REGION Network 14: PackML Event - Alarms Not Cleared
   RUNG wire#powerrail
      #instStatusAlarmsNotReset(EnableIn := wire#w1, Cfg_Event := "StatusCfg".Event[1], Cfg_MessagePrefix := "MessagePrefix".UN.Alarm, In_EventStatus := "UN".Status, Sts_Active => #instStatusAlarmsNotReset.Sts_Active, Sts_Latched => #instStatusAlarmsNotReset.Sts_Latched)
   END_RUNG
   RUNG wire#powerrail
      Contact( "PackML".Sts.State.Resetting )
      I_Contact( "UN".PackML_Sts_Alarm.sts_Resetting_SC )
   END_RUNG wire#w1
   RUNG wire#powerrail
      Contact( "PackML".Sts.State.Clearing )
      I_Contact( "UN".PackML_Sts_Alarm.sts_Clearing_SC )
   END_RUNG wire#w1
   // the same network as SCL:
   #instStatusAlarmsNotReset(EnableIn := ("PackML".Sts.State.Resetting AND NOT "UN".PackML_Sts_Alarm.sts_Resetting_SC) OR ("PackML".Sts.State.Clearing AND NOT "UN".PackML_Sts_Alarm.sts_Clearing_SC),   // "CPG_Event"
                           Cfg_Event := "StatusCfg".Event[1],
                           Cfg_MessagePrefix := "MessagePrefix".UN.Alarm,
                           In_EventStatus := "UN".Status,
                           Sts_Active => #instStatusAlarmsNotReset.Sts_Active,
                           Sts_Latched => #instStatusAlarmsNotReset.Sts_Latched);
END_REGION

REGION Network 15: Start Command
   // "PackTags".Command.CntrlCmd = 2 (start command value)
   RUNG wire#powerrail
      Contact( "PackML".remoteCommandEnable )
      { S7_Templates := "SrcType := DInt" } EQ_Contact(in1 := "PackTags".Command.CntrlCmd, in2 := "LPMLV30_CMD_START")
      Contact( "PackTags".Command.CmdChangeRequest )
      Coil( "UN".PackML_Sts_Alarm.cmd_Start )
   END_RUNG
   // the same network as SCL:
   "UN".PackML_Sts_Alarm.cmd_Start := "PackML".remoteCommandEnable AND ("PackTags".Command.CntrlCmd = "LPMLV30_CMD_START") AND "PackTags".Command.CmdChangeRequest;
END_REGION

REGION Network 16: Reset Command
   // "PackTags".Command.CntrlCmd = 1 (reset command value)
   RUNG wire#powerrail
      Contact( "PackML".remoteCommandEnable )
      { S7_Templates := "SrcType := DInt" } EQ_Contact(in1 := "PackTags".Command.CntrlCmd, in2 := "LPMLV30_CMD_RESET")
      Contact( "PackTags".Command.CmdChangeRequest )
      Coil( "UN".PackML_Sts_Alarm.cmd_Reset )
   END_RUNG
   // the same network as SCL:
   "UN".PackML_Sts_Alarm.cmd_Reset := "PackML".remoteCommandEnable AND ("PackTags".Command.CntrlCmd = "LPMLV30_CMD_RESET") AND "PackTags".Command.CmdChangeRequest;
END_REGION

REGION Network 17: Clear Command
   // "PackTags".Command.CntrlCmd = 9 (clear command value)
   RUNG wire#powerrail
      Contact( "PackML".remoteCommandEnable )
      { S7_Templates := "SrcType := DInt" } EQ_Contact(in1 := "PackTags".Command.CntrlCmd, in2 := "LPMLV30_CMD_CLEAR")
      Contact( "PackTags".Command.CmdChangeRequest )
      Coil( "UN".PackML_Sts_Alarm.cmd_Clear )
   END_RUNG
   // the same network as SCL:
   "UN".PackML_Sts_Alarm.cmd_Clear := "PackML".remoteCommandEnable AND ("PackTags".Command.CntrlCmd = "LPMLV30_CMD_CLEAR") AND "PackTags".Command.CmdChangeRequest;
END_REGION

REGION Network 18: *** EVENT CONTROL MANAGERS ***
END_REGION

REGION Network 19: Reset Command - for all event managers
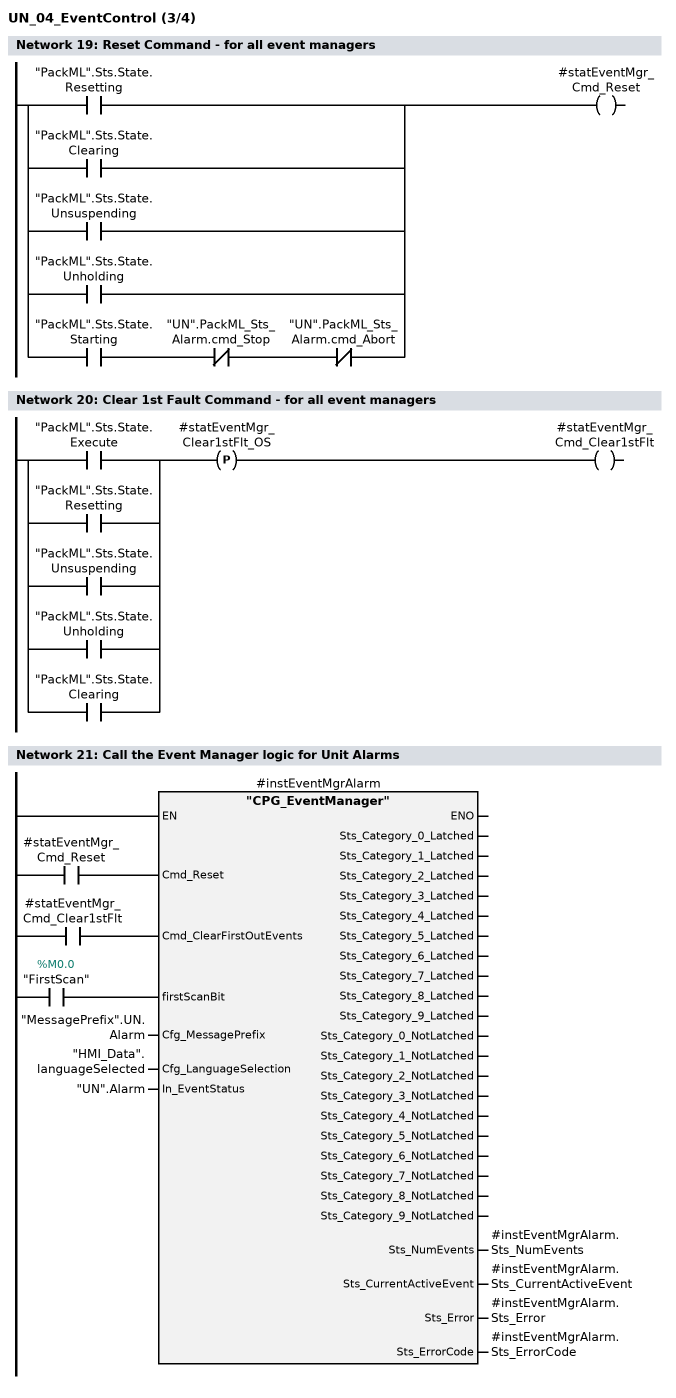
   RUNG wire#powerrail
      Contact( "PackML".Sts.State.Resetting )
      wire#w1
      Coil( #statEventMgr_Cmd_Reset )
   END_RUNG
   RUNG wire#powerrail
      Contact( "PackML".Sts.State.Clearing )
   END_RUNG wire#w1
   RUNG wire#powerrail
      Contact( "PackML".Sts.State.Unsuspending )
   END_RUNG wire#w1
   RUNG wire#powerrail
      Contact( "PackML".Sts.State.Unholding )
   END_RUNG wire#w1
   RUNG wire#powerrail
      Contact( "PackML".Sts.State.Starting )
      I_Contact( "UN".PackML_Sts_Alarm.cmd_Stop )
      I_Contact( "UN".PackML_Sts_Alarm.cmd_Abort )
   END_RUNG wire#w1
   // the same network as SCL:
   #statEventMgr_Cmd_Reset := "PackML".Sts.State.Resetting OR "PackML".Sts.State.Clearing OR "PackML".Sts.State.Unsuspending OR "PackML".Sts.State.Unholding OR ("PackML".Sts.State.Starting AND NOT "UN".PackML_Sts_Alarm.cmd_Stop AND NOT "UN".PackML_Sts_Alarm.cmd_Abort);
END_REGION

REGION Network 20: Clear 1st Fault Command - for all event managers
   RUNG wire#powerrail
      Contact( "PackML".Sts.State.Execute )
      wire#w1
      P_Trig( #statEventMgr_Clear1stFlt_OS )
      Coil( #statEventMgr_Cmd_Clear1stFlt )
   END_RUNG
   RUNG wire#powerrail
      Contact( "PackML".Sts.State.Resetting )
   END_RUNG wire#w1
   RUNG wire#powerrail
      Contact( "PackML".Sts.State.Unsuspending )
   END_RUNG wire#w1
   RUNG wire#powerrail
      Contact( "PackML".Sts.State.Unholding )
   END_RUNG wire#w1
   RUNG wire#powerrail
      Contact( "PackML".Sts.State.Clearing )
   END_RUNG wire#w1
   // the same network as SCL:
   #_w1 := "PackML".Sts.State.Execute OR "PackML".Sts.State.Resetting OR "PackML".Sts.State.Unsuspending OR "PackML".Sts.State.Unholding OR "PackML".Sts.State.Clearing;
   #_w2 := #_w1 AND NOT #statEventMgr_Clear1stFlt_OS;   // rising edge
   #statEventMgr_Clear1stFlt_OS := #_w1;
   #statEventMgr_Cmd_Clear1stFlt := #_w2;
END_REGION

REGION Network 21: Call the Event Manager logic for Unit Alarms
   RUNG wire#powerrail
      #instEventMgrAlarm(Cmd_Reset := wire#w1, Cmd_ClearFirstOutEvents := wire#w2, firstScanBit := wire#w3, Cfg_MessagePrefix := "MessagePrefix".UN.Alarm, Cfg_LanguageSelection := "HMI_Data".languageSelected, In_EventStatus := "UN".Alarm, Sts_Category_0_Latched =>, Sts_Category_1_Latched =>, Sts_Category_2_Latched =>, Sts_Category_3_Latched =>, Sts_Category_4_Latched =>, Sts_Category_5_Latched =>, Sts_Category_6_Latched =>, Sts_Category_7_Latched =>, Sts_Category_8_Latched =>, Sts_Category_9_Latched =>, Sts_Category_0_NotLatched =>, Sts_Category_1_NotLatched =>, Sts_Category_2_NotLatched =>, Sts_Category_3_NotLatched =>, Sts_Category_4_NotLatched =>, Sts_Category_5_NotLatched =>, Sts_Category_6_NotLatched =>, Sts_Category_7_NotLatched =>, Sts_Category_8_NotLatched =>, Sts_Category_9_NotLatched =>, Sts_NumEvents => #instEventMgrAlarm.Sts_NumEvents, Sts_CurrentActiveEvent => #instEventMgrAlarm.Sts_CurrentActiveEvent, Sts_Error => #instEventMgrAlarm.Sts_Error, Sts_ErrorCode => #instEventMgrAlarm.Sts_ErrorCode)
   END_RUNG
   RUNG wire#powerrail
      Contact( #statEventMgr_Cmd_Reset )
   END_RUNG wire#w1
   RUNG wire#powerrail
      Contact( #statEventMgr_Cmd_Clear1stFlt )
   END_RUNG wire#w2
   RUNG wire#powerrail
      Contact( "FirstScan" )
   END_RUNG wire#w3
   // the same network as SCL:
   #instEventMgrAlarm(Cmd_Reset := #statEventMgr_Cmd_Reset,   // "CPG_EventManager"
                      Cmd_ClearFirstOutEvents := #statEventMgr_Cmd_Clear1stFlt,
                      firstScanBit := "FirstScan",
                      Cfg_MessagePrefix := "MessagePrefix".UN.Alarm,
                      Cfg_LanguageSelection := "HMI_Data".languageSelected,
                      In_EventStatus := "UN".Alarm,
                      Sts_NumEvents => #instEventMgrAlarm.Sts_NumEvents,
                      Sts_CurrentActiveEvent => #instEventMgrAlarm.Sts_CurrentActiveEvent,
                      Sts_Error => #instEventMgrAlarm.Sts_Error,
                      Sts_ErrorCode => #instEventMgrAlarm.Sts_ErrorCode);
END_REGION

REGION Network 22: Call the Event Manager logic for Unit Warnings
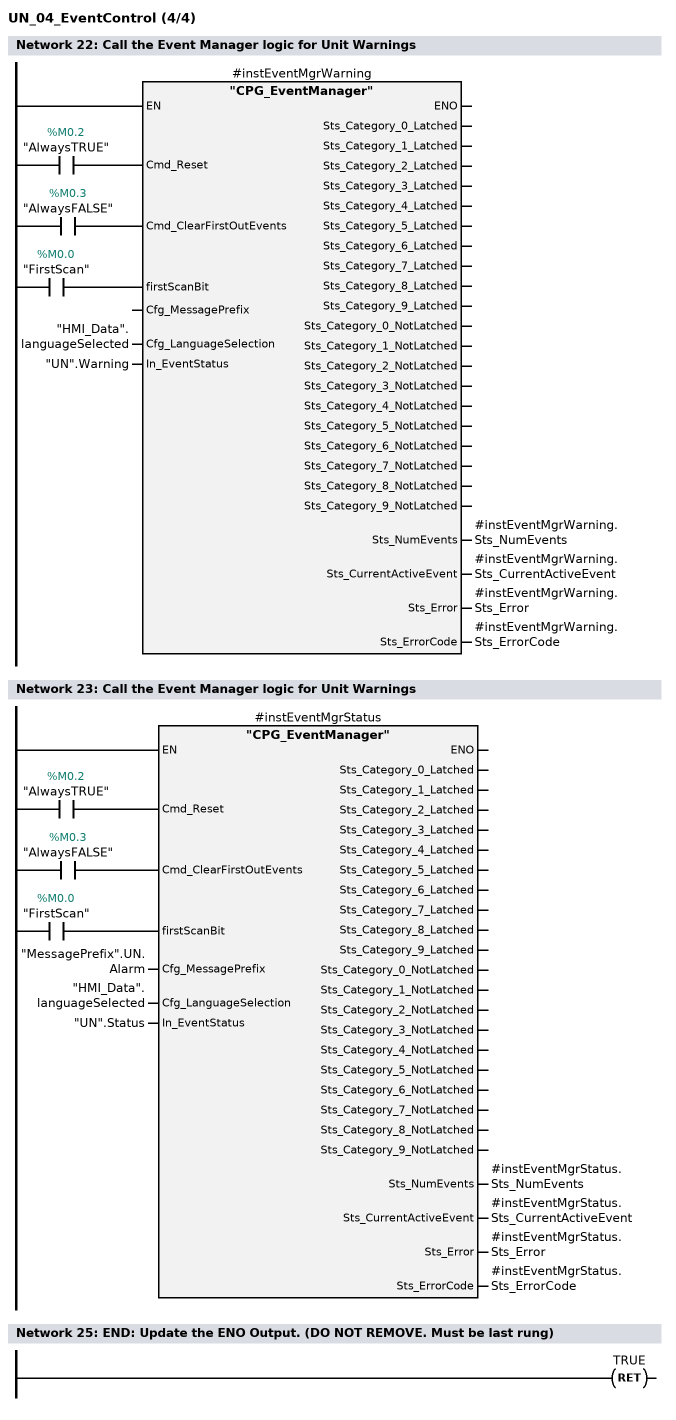
   RUNG wire#powerrail
      #instEventMgrWarning(Cmd_Reset := wire#w1, Cmd_ClearFirstOutEvents := wire#w2, firstScanBit := wire#w3, Cfg_MessagePrefix :=, Cfg_LanguageSelection := "HMI_Data".languageSelected, In_EventStatus := "UN".Warning, Sts_Category_0_Latched =>, Sts_Category_1_Latched =>, Sts_Category_2_Latched =>, Sts_Category_3_Latched =>, Sts_Category_4_Latched =>, Sts_Category_5_Latched =>, Sts_Category_6_Latched =>, Sts_Category_7_Latched =>, Sts_Category_8_Latched =>, Sts_Category_9_Latched =>, Sts_Category_0_NotLatched =>, Sts_Category_1_NotLatched =>, Sts_Category_2_NotLatched =>, Sts_Category_3_NotLatched =>, Sts_Category_4_NotLatched =>, Sts_Category_5_NotLatched =>, Sts_Category_6_NotLatched =>, Sts_Category_7_NotLatched =>, Sts_Category_8_NotLatched =>, Sts_Category_9_NotLatched =>, Sts_NumEvents => #instEventMgrWarning.Sts_NumEvents, Sts_CurrentActiveEvent => #instEventMgrWarning.Sts_CurrentActiveEvent, Sts_Error => #instEventMgrWarning.Sts_Error, Sts_ErrorCode => #instEventMgrWarning.Sts_ErrorCode)
   END_RUNG
   RUNG wire#powerrail
      Contact( "AlwaysTRUE" )
   END_RUNG wire#w1
   RUNG wire#powerrail
      Contact( "AlwaysFALSE" )
   END_RUNG wire#w2
   RUNG wire#powerrail
      Contact( "FirstScan" )
   END_RUNG wire#w3
   // the same network as SCL:
   #instEventMgrWarning(Cmd_Reset := "AlwaysTRUE",   // "CPG_EventManager"
                        Cmd_ClearFirstOutEvents := "AlwaysFALSE",
                        firstScanBit := "FirstScan",
                        Cfg_LanguageSelection := "HMI_Data".languageSelected,
                        In_EventStatus := "UN".Warning,
                        Sts_NumEvents => #instEventMgrWarning.Sts_NumEvents,
                        Sts_CurrentActiveEvent => #instEventMgrWarning.Sts_CurrentActiveEvent,
                        Sts_Error => #instEventMgrWarning.Sts_Error,
                        Sts_ErrorCode => #instEventMgrWarning.Sts_ErrorCode);
END_REGION

REGION Network 23: Call the Event Manager logic for Unit Warnings
   RUNG wire#powerrail
      #instEventMgrStatus(Cmd_Reset := wire#w1, Cmd_ClearFirstOutEvents := wire#w2, firstScanBit := wire#w3, Cfg_MessagePrefix := "MessagePrefix".UN.Alarm, Cfg_LanguageSelection := "HMI_Data".languageSelected, In_EventStatus := "UN".Status, Sts_Category_0_Latched =>, Sts_Category_1_Latched =>, Sts_Category_2_Latched =>, Sts_Category_3_Latched =>, Sts_Category_4_Latched =>, Sts_Category_5_Latched =>, Sts_Category_6_Latched =>, Sts_Category_7_Latched =>, Sts_Category_8_Latched =>, Sts_Category_9_Latched =>, Sts_Category_0_NotLatched =>, Sts_Category_1_NotLatched =>, Sts_Category_2_NotLatched =>, Sts_Category_3_NotLatched =>, Sts_Category_4_NotLatched =>, Sts_Category_5_NotLatched =>, Sts_Category_6_NotLatched =>, Sts_Category_7_NotLatched =>, Sts_Category_8_NotLatched =>, Sts_Category_9_NotLatched =>, Sts_NumEvents => #instEventMgrStatus.Sts_NumEvents, Sts_CurrentActiveEvent => #instEventMgrStatus.Sts_CurrentActiveEvent, Sts_Error => #instEventMgrStatus.Sts_Error, Sts_ErrorCode => #instEventMgrStatus.Sts_ErrorCode)
   END_RUNG
   RUNG wire#powerrail
      Contact( "AlwaysTRUE" )
   END_RUNG wire#w1
   RUNG wire#powerrail
      Contact( "AlwaysFALSE" )
   END_RUNG wire#w2
   RUNG wire#powerrail
      Contact( "FirstScan" )
   END_RUNG wire#w3
   // the same network as SCL:
   #instEventMgrStatus(Cmd_Reset := "AlwaysTRUE",   // "CPG_EventManager"
                       Cmd_ClearFirstOutEvents := "AlwaysFALSE",
                       firstScanBit := "FirstScan",
                       Cfg_MessagePrefix := "MessagePrefix".UN.Alarm,
                       Cfg_LanguageSelection := "HMI_Data".languageSelected,
                       In_EventStatus := "UN".Status,
                       Sts_NumEvents => #instEventMgrStatus.Sts_NumEvents,
                       Sts_CurrentActiveEvent => #instEventMgrStatus.Sts_CurrentActiveEvent,
                       Sts_Error => #instEventMgrStatus.Sts_Error,
                       Sts_ErrorCode => #instEventMgrStatus.Sts_ErrorCode);
END_REGION

REGION Network 25: END: Update the ENO Output. (DO NOT REMOVE. Must be last rung)
   RUNG wire#powerrail
      ReturnCoil( TRUE )
   END_RUNG
   // the same network as SCL:
   ENO := TRUE;
   RETURN;
END_REGION
END_FUNCTION_BLOCK

FUNCTION "CPG_ModuleInitialize" : Void
TITLE = CPG_ModuleInitialize
{ S7_Optimized_Access := 'TRUE' }
AUTHOR : 'tech.team.motioncontrol@siemens.com'
FAMILY : CPG
VERSION : 1.0
//Support: tech.team.motioncontrol@siemens.com
   VAR_INPUT 
      enableIn : Bool;   // Enable the FB call.
      firstScanBit : Bool;   // Bit used to tell logic that this is the first scan of PLC
   END_VAR

   VAR_IN_OUT 
      PackML_ModuleStatus : "CPG_typePackML_ModuleSts";   // PackML Module Status UDT
   END_VAR


BEGIN
	//============================================================================================================
	// SIEMENS AG
	// (c)Copyright 2018 All Rights Reserved
	//------------------------------------------------------------------------------------------------------------
	// Project: CPG Template
	// Tested with: S7-1500 with FW version V2.1
	// Engineering: TIA Portal V14
	// Restrictions: ---
	// Requirements: S7-1500
	// Functionality: This FC will initialize the "PackML" "Status" AND commands within a control module to ensure that the bits are in the correct state IF they are NOT being
	//                used later by that same control module. FOR example, if a start command is NOT being used by a control module, that bit should be turned off TO prevent
	//                unintentional starting OF the machine (in CASE it was accidentally OR through a rung edit turned on). IF a state complete bit FOR a particular state is
	//                NOT being used, that bit should be turned on TO allow the machine TO leave that state. This instruction is NOT needed FOR equipment modules OR the unit
	//                machine since all PackML status AND command bits are programmed in the summation routines.
	// Support: tech.team.motioncontrol@siemens.com
	//------------------------------------------------------------------------------------------------------------
	// Change log table:
	// Version       Date               Expert in charge    Changes applied
	//  01.00.00     01.01.2018         MP                  Initial Release & PackML V1.4  Renamed CPG V1.0
	//  01.01.00     22.05.2018         JP                  Adopted to styleguide
	//============================================================================================================
	// Function : CPG_ModuleInitialize
	//============================================================================================================
	
	
	(*  Command vs State Complete:
	•   State complete bits are AND’d together, meaning that all control modules and equipment modules must be done with an acting state 
	      before it can transition to the wait state. For example, all of the CM’s and EM’s must be done Stopping before the machine can 
	      transition to the Stopped state.
	•   With two exceptions, PackML commands (such as Start, Stop, Abort, Suspend, etc.) are OR’d together, meaning that any 1 control or 
	      equipment module can cause the machine to initiate action.  For example, the Stop command initiated from 1 equipment module will 
	      stop the entire machine.  
	
	The only exceptions to this rule are the PackML commands UnHold and UnSuspend.  In either case, the UnHold and UnSuspend commands act 
	      like state complete bits.  By doing this in a modular machine architecture, this prevents 1 equipment module from sending the 
	      machine into UnHolding or UnSuspending when another equipment module is still wanting the machine to stay held or suspended.  
	      For example, assume that both the Infeed Equipment Module (Starved) and Discharge Equipment Module (Blocked) is telling the 
	      machine to suspend, if the Infeed Equipment Module has product again, the machine should not UnSuspend without the Discharge 
	      Equipment Module also becoming unblocked.
	*)
	
	IF #firstScanBit OR #enableIn THEN
	// Reset all Command (CMD) bits - this forces the command(CMD) bit to be set in user program if the command is required/used by the CM
	    #PackML_ModuleStatus.cmd_Reset           := FALSE; //
	    #PackML_ModuleStatus.cmd_Start           := FALSE; //
	    #PackML_ModuleStatus.cmd_Stop            := FALSE; //
	    #PackML_ModuleStatus.cmd_Hold            := FALSE; //
	    #PackML_ModuleStatus.cmd_Suspend         := FALSE; //
	    #PackML_ModuleStatus.cmd_Abort           := FALSE; //
	    #PackML_ModuleStatus.cmd_Clear           := FALSE; //
	
	// Set all State Complete (SC) bits - setting the SC bit true allows CM to transition to the next step with no user code need. If the
	// respective SC bit is used by the CM, then user logic must be added to set/reset SC bits as required by the application.
	    #PackML_ModuleStatus.sts_Resetting_SC    := TRUE; //
	    #PackML_ModuleStatus.sts_Starting_SC     := TRUE; //
	    #PackML_ModuleStatus.sts_Stopping_SC     := TRUE; //
	    #PackML_ModuleStatus.sts_Holding_SC      := TRUE; //
	    #PackML_ModuleStatus.sts_UnHolding_SC    := TRUE; //
	    #PackML_ModuleStatus.sts_Suspending_SC   := TRUE; //
	    #PackML_ModuleStatus.sts_UnSuspending_SC := TRUE; //
	    #PackML_ModuleStatus.sts_Aborting_SC     := TRUE; //
	    #PackML_ModuleStatus.sts_Clearing_SC     := TRUE; //
	    #PackML_ModuleStatus.sts_Execute_SC      := TRUE; //
	    #PackML_ModuleStatus.sts_Completing_SC   := TRUE; //
	
	    //
	    #PackML_ModuleStatus.cmd_UnHold          := TRUE; //
	    #PackML_ModuleStatus.cmd_UnSuspend       := TRUE; //
	
	END_IF;  // End "IF FirstScanBit OR EnableIn THEN"
	
	//  -------------- END OF LOGIC -------------------------
	ENO := TRUE;   // Set the ENO output
	
END_FUNCTION

FUNCTION_BLOCK "CPG_EventManager"
TITLE = CPG_EventManager
{ S7_Optimized_Access := 'TRUE' }
AUTHOR : 'tech.team.motioncontrol@siemens.com'
FAMILY : CPG
VERSION : 1.0
//Support: tech.team.motioncontrol@siemens.com
   VAR_INPUT 
      Cmd_Reset { ExternalAccessible := 'False'; ExternalVisible := 'False'; ExternalWritable := 'False'} : Bool;   // Reset Command
      Cmd_ClearFirstOutEvents { ExternalAccessible := 'False'; ExternalVisible := 'False'; ExternalWritable := 'False'} : Bool;   // Command to clear First Out events
      firstScanBit { ExternalAccessible := 'False'; ExternalVisible := 'False'; ExternalWritable := 'False'} : Bool;   // Bit used to tell logic that this is the first scan of PLC
      Cfg_MessagePrefix { ExternalAccessible := 'False'; ExternalVisible := 'False'; ExternalWritable := 'False'} : "CPG_typeMessagePrefix";   // Message Prefix value for event messages multi-lingual
      Cfg_LanguageSelection { ExternalAccessible := 'False'; ExternalVisible := 'False'; ExternalWritable := 'False'} : Int;   // Current Langage: 0=EN, 1=DE, 2=SP/ES, 3=IT, 4=FR
   END_VAR

   VAR_OUTPUT 
      Sts_Category_0_Latched { ExternalAccessible := 'False'; ExternalVisible := 'False'; ExternalWritable := 'False'; S7_HiddenAssignment := 'HideIfNoParamAssigned'} : Bool;   // Event Category Status (on until reset cmd) - CAT 0
      Sts_Category_1_Latched { ExternalAccessible := 'False'; ExternalVisible := 'False'; ExternalWritable := 'False'; S7_HiddenAssignment := 'HideIfNoParamAssigned'} : Bool;   // Event Category Status (on until reset cmd) - CAT 1
      Sts_Category_2_Latched { ExternalAccessible := 'False'; ExternalVisible := 'False'; ExternalWritable := 'False'; S7_HiddenAssignment := 'HideIfNoParamAssigned'} : Bool;   // Event Category Status (on until reset cmd) - CAT 2
      Sts_Category_3_Latched { ExternalAccessible := 'False'; ExternalVisible := 'False'; ExternalWritable := 'False'; S7_HiddenAssignment := 'HideIfNoParamAssigned'} : Bool;   // Event Category Status (on until reset cmd) - CAT 3
      Sts_Category_4_Latched { ExternalAccessible := 'False'; ExternalVisible := 'False'; ExternalWritable := 'False'; S7_HiddenAssignment := 'HideIfNoParamAssigned'} : Bool;   // Event Category Status (on until reset cmd) - CAT 4
      Sts_Category_5_Latched { ExternalAccessible := 'False'; ExternalVisible := 'False'; ExternalWritable := 'False'; S7_HiddenAssignment := 'HideIfNoParamAssigned'} : Bool;   // Event Category Status (on until reset cmd) - CAT 5
      Sts_Category_6_Latched { ExternalAccessible := 'False'; ExternalVisible := 'False'; ExternalWritable := 'False'; S7_HiddenAssignment := 'HideIfNoParamAssigned'} : Bool;   // Event Category Status (on until reset cmd) - CAT 6
      Sts_Category_7_Latched { ExternalAccessible := 'False'; ExternalVisible := 'False'; ExternalWritable := 'False'; S7_HiddenAssignment := 'HideIfNoParamAssigned'} : Bool;   // Event Category Status (on until reset cmd) - CAT 7
      Sts_Category_8_Latched { ExternalAccessible := 'False'; ExternalVisible := 'False'; ExternalWritable := 'False'; S7_HiddenAssignment := 'HideIfNoParamAssigned'} : Bool;   // Event Category Status (on until reset cmd) - CAT 8
      Sts_Category_9_Latched { ExternalAccessible := 'False'; ExternalVisible := 'False'; ExternalWritable := 'False'; S7_HiddenAssignment := 'HideIfNoParamAssigned'} : Bool;   // Event Category Status (on until reset cmd) - CAT 9
      Sts_Category_0_NotLatched { ExternalAccessible := 'False'; ExternalVisible := 'False'; ExternalWritable := 'False'; S7_HiddenAssignment := 'HideIfNoParamAssigned'} : Bool;   // Event Cat Status, not latched (=active event status) - CAT 0
      Sts_Category_1_NotLatched { ExternalAccessible := 'False'; ExternalVisible := 'False'; ExternalWritable := 'False'; S7_HiddenAssignment := 'HideIfNoParamAssigned'} : Bool;   // Event Cat Status, not latched (=active event status) - CAT 1
      Sts_Category_2_NotLatched { ExternalAccessible := 'False'; ExternalVisible := 'False'; ExternalWritable := 'False'; S7_HiddenAssignment := 'HideIfNoParamAssigned'} : Bool;   // Event Cat Status, not latched (=active event status) - CAT 2
      Sts_Category_3_NotLatched { ExternalAccessible := 'False'; ExternalVisible := 'False'; ExternalWritable := 'False'; S7_HiddenAssignment := 'HideIfNoParamAssigned'} : Bool;   // Event Cat Status, not latched (=active event status) - CAT 3
      Sts_Category_4_NotLatched { ExternalAccessible := 'False'; ExternalVisible := 'False'; ExternalWritable := 'False'; S7_HiddenAssignment := 'HideIfNoParamAssigned'} : Bool;   // Event Cat Status, not latched (=active event status) - CAT 4
      Sts_Category_5_NotLatched { ExternalAccessible := 'False'; ExternalVisible := 'False'; ExternalWritable := 'False'; S7_HiddenAssignment := 'HideIfNoParamAssigned'} : Bool;   // Event Cat Status, not latched (=active event status) - CAT 5
      Sts_Category_6_NotLatched { ExternalAccessible := 'False'; ExternalVisible := 'False'; ExternalWritable := 'False'; S7_HiddenAssignment := 'HideIfNoParamAssigned'} : Bool;   // Event Cat Status, not latched (=active event status) - CAT 6
      Sts_Category_7_NotLatched { ExternalAccessible := 'False'; ExternalVisible := 'False'; ExternalWritable := 'False'; S7_HiddenAssignment := 'HideIfNoParamAssigned'} : Bool;   // Event Cat Status, not latched (=active event status) - CAT 7
      Sts_Category_8_NotLatched { ExternalAccessible := 'False'; ExternalVisible := 'False'; ExternalWritable := 'False'; S7_HiddenAssignment := 'HideIfNoParamAssigned'} : Bool;   // Event Cat Status, not latched (=active event status) - CAT 8
      Sts_Category_9_NotLatched { ExternalAccessible := 'False'; ExternalVisible := 'False'; ExternalWritable := 'False'; S7_HiddenAssignment := 'HideIfNoParamAssigned'} : Bool;   // Event Cat Status, not latched (=active event status) - CAT 9
      Sts_NumEvents { ExternalAccessible := 'False'; ExternalVisible := 'False'; ExternalWritable := 'False'} : Int;   // Number of event in the In_EventStatus list
      Sts_CurrentActiveEvent { ExternalAccessible := 'False'; ExternalVisible := 'False'; ExternalWritable := 'False'} : Bool;   // Status - TRUE = if any active events
      Sts_Error { ExternalAccessible := 'False'; ExternalVisible := 'False'; ExternalWritable := 'False'} : Bool;   // FB Error exist
      Sts_ErrorCode { ExternalAccessible := 'False'; ExternalVisible := 'False'; ExternalWritable := 'False'} : DInt;   // FB Error code
   END_VAR

   VAR_IN_OUT 
      In_EventStatus : "CPG_typeEventStatus";   // Working event list data section
   END_VAR

   VAR 
      statEventCategory { ExternalAccessible := 'False'; ExternalVisible := 'False'; ExternalWritable := 'False'} : DInt;
      statIndexAllEvents { ExternalAccessible := 'False'; ExternalVisible := 'False'; ExternalWritable := 'False'} : Int;
      statIndexClearActiveEvents { ExternalAccessible := 'False'; ExternalVisible := 'False'; ExternalWritable := 'False'} : Int;
      statIndexClearFirstOut { ExternalAccessible := 'False'; ExternalVisible := 'False'; ExternalWritable := 'False'} : Int;
      statNumEvents { ExternalAccessible := 'False'; ExternalVisible := 'False'; ExternalWritable := 'False'} : Int;   // Max # of Events
      statPrevCmdReset { ExternalAccessible := 'False'; ExternalVisible := 'False'; ExternalWritable := 'False'} : Bool;
      statPrevNumEvents { ExternalAccessible := 'False'; ExternalVisible := 'False'; ExternalWritable := 'False'} : Int;
      statPrevUpdateEventListID { ExternalAccessible := 'False'; ExternalVisible := 'False'; ExternalWritable := 'False'} : Int;
      statUpdateEventList { ExternalAccessible := 'False'; ExternalVisible := 'False'; ExternalWritable := 'False'} : Bool;
      statCurrentErrorCode { ExternalAccessible := 'False'; ExternalVisible := 'False'; ExternalWritable := 'False'} : Int;
      statCurrentActiveEvent { ExternalAccessible := 'False'; ExternalVisible := 'False'; ExternalWritable := 'False'} : Bool;
      statZeroEvent { ExternalAccessible := 'False'; ExternalVisible := 'False'; ExternalWritable := 'False'} : "CPG_typeEvent";   // Null Event
   END_VAR


BEGIN
	//============================================================================================================
	// SIEMENS AG
	// (c)Copyright 2018 All Rights Reserved
	//------------------------------------------------------------------------------------------------------------
	// Project: CPG Template
	// Tested with: S7-1500 with FW version V2.1
	// Engineering: TIA Portal V14
	// Restrictions: ---
	// Requirements: S7-1500
	// Functionality: Control EventManager function
	// Support: tech.team.motioncontrol@siemens.com
	//------------------------------------------------------------------------------------------------------------
	// Change log table:
	// Version       Date               Expert in charge    Changes applied
	//  01.00.00     01.01.2018         MP                  Initial Release & PackML V1.8  Renamed CPG V1.0
	//  01.01.00     22.05.2018         JP                  Adopted to styleguide
	//============================================================================================================
	// Function : CPG_EventManager
	//============================================================================================================
	
	// First Scan Logic Logic (only run through on 1st scan of PLC)
	IF #firstScanBit THEN                                                                   // Only run first scan
	  #In_EventStatus.wrk_ResetID := #In_EventStatus.wrk_ResetID + 1;                     // increment the Work Reset ID
	  #In_EventStatus.wrk_UpdateEventListID := #In_EventStatus.wrk_UpdateEventListID + 1; // increment the Work UpdateList ID
	  #In_EventStatus.sts_NumAllEvents := 0;                                              // Reset the number of all events value
	  
	  // Determine the Number of Sts_Events for given alarm/warning area
	  "CPG_ArrayLength"(arrayToBeSized := #In_EventStatus.sts_Events,
	                    arraySize => #In_EventStatus.wrk_EventArraySize);
	  RETURN;     // Exit the FB call
	END_IF;         // End the first scan section
	
	
	//---------------------------------------------------------------------------------
	// Main Logic Section
	
	// Update the message prefix for the current language
	IF #Cfg_LanguageSelection >= 0 AND #Cfg_LanguageSelection <= "LPMLV30_LANGUAGES_UPPER_LIM" THEN
	  #In_EventStatus.wrk_MessagePrefix := #Cfg_MessagePrefix.messagePrefix[#Cfg_LanguageSelection];
	END_IF;
	#In_EventStatus.wrk_LanguageSelection := #Cfg_LanguageSelection;
	
	// Upon a reset command, reset the latched status bits and clear the event list
	IF #Cmd_Reset THEN
	  #In_EventStatus.sts_Category_0_Latched := FALSE;
	  #In_EventStatus.sts_Category_1_Latched := FALSE;
	  #In_EventStatus.sts_Category_2_Latched := FALSE;
	  #In_EventStatus.sts_Category_3_Latched := FALSE;
	  #In_EventStatus.sts_Category_4_Latched := FALSE;
	  #In_EventStatus.sts_Category_5_Latched := FALSE;
	  #In_EventStatus.sts_Category_6_Latched := FALSE;
	  #In_EventStatus.sts_Category_7_Latched := FALSE;
	  #In_EventStatus.sts_Category_8_Latched := FALSE;
	  #In_EventStatus.sts_Category_9_Latched := FALSE;
	  
	  IF NOT (#statPrevCmdReset) THEN                             // Clear the zero event
	    #In_EventStatus.out_ZeroEvent := #statZeroEvent;
	    // String seperation variable not added.
	  END_IF;
	END_IF;                      // End IF Cmd_Reset.... 
	
	
	// Clear first out events - for alarms, this is typically done once the machine starts    
	IF #Cmd_ClearFirstOutEvents AND NOT (#statCurrentActiveEvent) THEN
	  #In_EventStatus.sts_FirstOutEvent := #In_EventStatus.out_ZeroEvent;
	  
	  FOR #statIndexClearFirstOut := 0 TO 9 BY 1 DO
	    #In_EventStatus.sts_FirstOutEventCat[#statIndexClearFirstOut] := #In_EventStatus.out_ZeroEvent;
	  END_FOR;
	END_IF;
	
	// Determine the maximum number of event that can be stored in the array.
	// It is assumed that the input array size is equal to the output array size
	IF (#Cmd_Reset AND (NOT #statPrevCmdReset)) OR (#In_EventStatus.wrk_EventArraySize = 0) THEN
	  // Determine the Number of Sts_Events for given alarm/warning area
	  
	  "CPG_ArrayLength"(arrayToBeSized := #In_EventStatus.sts_Events,
	                    arraySize => #In_EventStatus.wrk_EventArraySize);
	END_IF;
	
	//Determine if the event list needs updating    
	IF #In_EventStatus.wrk_UpdateEventListID <> #statPrevUpdateEventListID THEN
	  #statPrevUpdateEventListID := #In_EventStatus.wrk_UpdateEventListID;
	  #statUpdateEventList := TRUE;
	END_IF;
	
	IF #statUpdateEventList THEN
	  #statUpdateEventList := FALSE;
	  // Update Event outputs and status
	  // First clear the not latched staus bits and total number of events.
	  // This instruction will find the events in the coming rungs
	  #statCurrentErrorCode := 0;
	  #Sts_NumEvents := #In_EventStatus.sts_NumAllEvents;
	  #statCurrentActiveEvent := FALSE;
	  #Sts_Category_0_NotLatched := FALSE;
	  #Sts_Category_1_NotLatched := FALSE;
	  #Sts_Category_2_NotLatched := FALSE;
	  #Sts_Category_3_NotLatched := FALSE;
	  #Sts_Category_4_NotLatched := FALSE;
	  #Sts_Category_5_NotLatched := FALSE;
	  #Sts_Category_6_NotLatched := FALSE;
	  #Sts_Category_7_NotLatched := FALSE;
	  #Sts_Category_8_NotLatched := FALSE;
	  #Sts_Category_9_NotLatched := FALSE;
	  
	  //Determine if the number of events is greater than the max array size        
	  //if so, then report error
	  #statNumEvents := #In_EventStatus.sts_NumAllEvents;
	  IF #statNumEvents > #In_EventStatus.wrk_EventArraySize THEN
	    #statNumEvents := #In_EventStatus.wrk_EventArraySize;
	    IF (#statCurrentErrorCode = 0) THEN                   // Update status error code
	      #statCurrentErrorCode := 1;
	    END_IF;
	  END_IF;
	  #In_EventStatus.sts_NumEvents := #statNumEvents;
	  
	  //Go through the event array to capture first fault event and perform string management        
	  #statIndexAllEvents := 0;
	  FOR #statIndexAllEvents := 0 TO #statNumEvents - 1 DO
	    // Check to see if any event is currently still active
	    IF (#In_EventStatus.sts_Events[#statIndexAllEvents].Trigger) THEN
	      #statCurrentActiveEvent := TRUE;
	    END_IF;
	    
	    //Store event category for logic later in code
	    IF (#In_EventStatus.sts_Events[#statIndexAllEvents].Category >= 0) AND (#In_EventStatus.sts_Events[#statIndexAllEvents].Category <= 9) THEN
	      #statEventCategory := #In_EventStatus.sts_Events[#statIndexAllEvents].Category;
	    ELSE
	      #statEventCategory := 0;
	      IF (#statCurrentErrorCode = 0) THEN                   // Update status error code
	        #statCurrentErrorCode := 2;
	      END_IF;         // end "IF (Sts_ErrorCode=0)"
	    END_IF;             // end "IF (In_EventStatus.Sts_Events[Inde..."    
	    
	    // Set the First Out Event
	    IF NOT (#In_EventStatus.sts_FirstOutEvent.Trigger) THEN
	      #In_EventStatus.sts_FirstOutEvent := #In_EventStatus.sts_Events[#statIndexAllEvents];
	      #In_EventStatus.sts_FirstOutEvent.Trigger := TRUE;
	    END_IF;
	    
	    // Set the First Out Events by category
	    IF NOT (#In_EventStatus.sts_FirstOutEventCat[#statEventCategory].Trigger) THEN
	      #In_EventStatus.sts_FirstOutEventCat[#statEventCategory] := #In_EventStatus.sts_Events[#statIndexAllEvents];
	      #In_EventStatus.sts_FirstOutEventCat[#statEventCategory].Trigger := TRUE;
	    END_IF;
	    
	    //Category Event Status            
	    CASE DINT_TO_INT(#In_EventStatus.sts_Events[#statIndexAllEvents].Category) OF
	      0:
	        #Sts_Category_0_NotLatched := #In_EventStatus.sts_Events[#statIndexAllEvents].Trigger;
	      1:
	        #Sts_Category_1_NotLatched := (#Sts_Category_1_NotLatched OR #In_EventStatus.sts_Events[#statIndexAllEvents].Trigger);
	      2:
	        #Sts_Category_2_NotLatched := (#Sts_Category_2_NotLatched OR #In_EventStatus.sts_Events[#statIndexAllEvents].Trigger);
	      3:
	        #Sts_Category_3_NotLatched := (#Sts_Category_3_NotLatched OR #In_EventStatus.sts_Events[#statIndexAllEvents].Trigger);
	      4:
	        #Sts_Category_4_NotLatched := (#Sts_Category_4_NotLatched OR #In_EventStatus.sts_Events[#statIndexAllEvents].Trigger);
	      5:
	        #Sts_Category_5_NotLatched := (#Sts_Category_5_NotLatched OR #In_EventStatus.sts_Events[#statIndexAllEvents].Trigger);
	      6:
	        #Sts_Category_6_NotLatched := (#Sts_Category_6_NotLatched OR #In_EventStatus.sts_Events[#statIndexAllEvents].Trigger);
	      7:
	        #Sts_Category_7_NotLatched := (#Sts_Category_7_NotLatched OR #In_EventStatus.sts_Events[#statIndexAllEvents].Trigger);
	      8:
	        #Sts_Category_8_NotLatched := (#Sts_Category_8_NotLatched OR #In_EventStatus.sts_Events[#statIndexAllEvents].Trigger);
	      9:
	        #Sts_Category_9_NotLatched := (#Sts_Category_9_NotLatched OR #In_EventStatus.sts_Events[#statIndexAllEvents].Trigger);
	    END_CASE;  // End of DINT_TO_INT(In_EventStatus.sts_events[Ind....
	    
	    
	  END_FOR;
	  
	  // set the status bits
	  #Sts_Category_0_Latched := #In_EventStatus.sts_Category_0_Latched;
	  #Sts_Category_1_Latched := #In_EventStatus.sts_Category_1_Latched;
	  #Sts_Category_2_Latched := #In_EventStatus.sts_Category_2_Latched;
	  #Sts_Category_3_Latched := #In_EventStatus.sts_Category_3_Latched;
	  #Sts_Category_4_Latched := #In_EventStatus.sts_Category_4_Latched;
	  #Sts_Category_5_Latched := #In_EventStatus.sts_Category_5_Latched;
	  #Sts_Category_6_Latched := #In_EventStatus.sts_Category_6_Latched;
	  #Sts_Category_7_Latched := #In_EventStatus.sts_Category_7_Latched;
	  #Sts_Category_8_Latched := #In_EventStatus.sts_Category_8_Latched;
	  #Sts_Category_9_Latched := #In_EventStatus.sts_Category_9_Latched;
	  
	  #In_EventStatus.sts_Category_0_NotLatched := #Sts_Category_0_NotLatched;
	  #In_EventStatus.sts_Category_1_NotLatched := #Sts_Category_1_NotLatched;
	  #In_EventStatus.sts_Category_2_NotLatched := #Sts_Category_2_NotLatched;
	  #In_EventStatus.sts_Category_3_NotLatched := #Sts_Category_3_NotLatched;
	  #In_EventStatus.sts_Category_4_NotLatched := #Sts_Category_4_NotLatched;
	  #In_EventStatus.sts_Category_5_NotLatched := #Sts_Category_5_NotLatched;
	  #In_EventStatus.sts_Category_6_NotLatched := #Sts_Category_6_NotLatched;
	  #In_EventStatus.sts_Category_7_NotLatched := #Sts_Category_7_NotLatched;
	  #In_EventStatus.sts_Category_8_NotLatched := #Sts_Category_8_NotLatched;
	  #In_EventStatus.sts_Category_9_NotLatched := #Sts_Category_9_NotLatched;
	  
	  #In_EventStatus.sts_CurrentActiveEvent := #statCurrentActiveEvent;
	END_IF;
	
	// Clear the remaining inactive bits    
	IF #statPrevNumEvents > #In_EventStatus.sts_NumEvents THEN
	  FOR #statIndexClearActiveEvents := #In_EventStatus.sts_NumEvents TO #statPrevNumEvents - 1 DO
	    #In_EventStatus.sts_Events[#statIndexClearActiveEvents] := #In_EventStatus.out_ZeroEvent;
	  END_FOR;
	END_IF;
	
	// Clear the number of input events in the case where some control module events are not being actively scanned.    
	IF #Cmd_Reset AND ((#In_EventStatus.sts_CurrentActiveEvent) OR (#In_EventStatus.sts_NumEvents > 0) OR (NOT #statPrevCmdReset)) THEN
	  #In_EventStatus.wrk_ResetID := #In_EventStatus.wrk_ResetID + 1;
	  #In_EventStatus.wrk_UpdateEventListID := #In_EventStatus.wrk_UpdateEventListID + 1;
	  #In_EventStatus.sts_NumAllEvents := 0;
	END_IF;
	
	#statPrevNumEvents := #In_EventStatus.sts_NumEvents;
	#statPrevCmdReset := #Cmd_Reset;
	
	//Write outputs
	#Sts_ErrorCode := #statCurrentErrorCode;
	#Sts_Error := (#statCurrentErrorCode <> 0);
	#Sts_CurrentActiveEvent := #statCurrentActiveEvent;
	
	//-----------------------------------------------------
	ENO := TRUE;   // Set the ENO output
	
END_FUNCTION_BLOCK

FUNCTION "CPG_ArrayLength" : Void
TITLE = CPG_ArrayLength
{ S7_Optimized_Access := 'TRUE' }
AUTHOR : 'tech.team.motioncontrol@siemens.com'
FAMILY : CPG
VERSION : 1.0
//Support: tech.team.motioncontrol@siemens.com
   VAR_INPUT 
      arrayToBeSized : Variant;   // Array to be sized
   END_VAR

   VAR_OUTPUT 
      arraySize : Int;   // Number of elements (size) in an array
   END_VAR


BEGIN
	//============================================================================================================
	// SIEMENS AG
	// (c)Copyright 2018 All Rights Reserved
	//------------------------------------------------------------------------------------------------------------
	// Project: CPG Template
	// Tested with: S7-1500 with FW version V2.1
	// Engineering: TIA Portal V14
	// Restrictions: ---
	// Requirements: S7-1x00
	// Functionality: Function Call to determine the length of any array
	//                using optimized S7-1x00 Data Blocks (DB).
	//                This FC can be called from any other FC/FB using any programming
	//                language (SCL, LAD).  Additionally it works with Firmware >= V1.8 
	//                and can determine the size of arrays with elementary (INT,Bool, etc.)
	//                or complex data types (structures)
	// Support: tech.team.motioncontrol@siemens.com
	//------------------------------------------------------------------------------------------------------------
	// Change log table:
	// Version       Date               Expert in charge    Changes applied
	//  01.00.00     08.12.2014         MP                  Initial Release 
	//  01.01.00     22.05.2018         JP                  Adopted to styleguide
	//============================================================================================================
	// Function : CPG_ArrayLength
	//============================================================================================================
	
	
	IF IS_ARRAY(#arrayToBeSized) THEN // Check if input is valid array
	  #arraySize := UDINT_TO_INT(CountOfElements(#arrayToBeSized)); // Determine the length of the array
	END_IF;
	
	ENO := TRUE;   // Set the ENO output
END_FUNCTION

FUNCTION_BLOCK "UN_05_EventSummation"   // FB31625, LAD
TITLE = UN_05_EventSummation
{ S7_Optimized_Access := 'TRUE' }
AUTHOR : tech.team.motioncontrol@siemens.com
FAMILY : CPG
VERSION : 1.1
// Support: tech.team.motioncontrol@siemens.com
// stored: AutoNumber true, IsIECCheckEnabled false, IsRetainMemResEnabled false, MemoryReserve 100, SetENOAutomatically false, UDAEnableTagReadback false
   VAR
      instEventSumBeg_Alarm { S7_SetPoint := 'True'} : "CPG_EventSummationBegin";   // instanceFB - EventSummationBegin - Alarm Events
      instEventSum_Alarm_UN { S7_SetPoint := 'True'} : "CPG_EventSummation";   // instanceFB - EventSummation FB - Alarm Events - UN
      instEventSum_Alarm_EM00 { S7_SetPoint := 'True'} : "CPG_EventSummation";   // instanceFB - EventSummation FB - Alarm Events - EM00
      instEventSum_Alarm_EM01 { S7_SetPoint := 'True'} : "CPG_EventSummation";   // instanceFB - EventSummation FB - Alarm Events - EM01
      instEventSum_Alarm_EM02 { S7_SetPoint := 'True'} : "CPG_EventSummation";   // instanceFB - EventSummation FB - Alarm Events - EM02
      instEventSumEnd_Alarm { S7_SetPoint := 'True'} : "CPG_EventSummationEnd";   // instanceFB - EventSummationEnd - Alarm Events
      instEventSortFilter_Alarm { S7_SetPoint := 'True'} : "CPG_EventSortFilter";   // instanceFB - EventSortFilter FB - Alarms
      instAlarmMove { S7_SetPoint := 'True'} : "CPG_AlarmMove";   // instance FB - Alarm Move
      instEventSumBeg_Warning { S7_SetPoint := 'True'} : "CPG_EventSummationBegin";   // instanceFB - EventSummationBegin - Warning Events
      instEventSum_Warning_UN { S7_SetPoint := 'True'} : "CPG_EventSummation";   // instanceFB - EventSummation FB - Warning Events - UN
      instEventSum_Warning_EM00 { S7_SetPoint := 'True'} : "CPG_EventSummation";   // instanceFB - EventSummation FB - Warning Events - EM00
      instEventSum_Warning_EM01 { S7_SetPoint := 'True'} : "CPG_EventSummation";   // instanceFB - EventSummation FB - Warning Events - EM01
      instEventSum_Warning_EM02 { S7_SetPoint := 'True'} : "CPG_EventSummation";   // instanceFB - EventSummation FB - Warning Events - EM02
      instEventSumEnd_Warning { S7_SetPoint := 'True'} : "CPG_EventSummationEnd";   // instanceFB - EventSummationEnd - Warning Events
      instEventSortFilter_Warning { S7_SetPoint := 'True'} : "CPG_EventSortFilter";   // instanceFB - EventSortFilter FB - Alarms
      instWarning_MsgScroll { S7_SetPoint := 'True'} : "CPG_MsgScroll";   // instance FB - Warning Scroll
      instEventSumBeg_Status { S7_SetPoint := 'True'} : "CPG_EventSummationBegin";   // instanceFB - EventSummationBegin - Status Events
      instEventSum_Status_UN { S7_SetPoint := 'True'} : "CPG_EventSummation";   // instanceFB - EventSummation FB - Status Events - UN
      instEventSum_Status_EM00 { S7_SetPoint := 'True'} : "CPG_EventSummation";   // instanceFB - EventSummation FB - Status Events - EM00
      instEventSum_Status_EM01 { S7_SetPoint := 'True'} : "CPG_EventSummation";   // instanceFB - EventSummation FB - Status Events - EM01
      instEventSum_Status_EM02 { S7_SetPoint := 'True'} : "CPG_EventSummation";   // instanceFB - EventSummation FB - Status Events - EM02
      instEventSumEnd_Status { S7_SetPoint := 'True'} : "CPG_EventSummationEnd";   // instanceFB - EventSummationEnd - Status Events
      instPackML_AlarmHistory { S7_SetPoint := 'True'} : "CPG_AlarmHistory";   // instance FB - Capturing the 1st fault history
      instProgram_Alarm { S7_SetPoint := 'True'} : Program_Alarm;   // instance DB for Program Alarm - diag to PLC HMI
      instWarningMove { S7_SetPoint := 'True'} : "CPG_AlarmMove";
      instPareto { S7_SetPoint := 'True'} : "CPG_ParetoAnalysis";
   END_VAR
   VAR_TEMP
      tempAlarmMove_Sts_Error : Bool;   // Error with AlarmMove?
      tempAlarmMove_Sts_ErrorCode : Int;   // AlarmMove Error code
      tempProgramAlarm_error : Bool;
      tempProgramAlarm_status : Word;
   END_VAR
BEGIN

REGION Network 1: Call the Alarm Event Summary - Beginning FB
   // **********  ALARM CONTROL SUMMATION  **********
   //  
   // The event summation begin instruction prepares the summation blocks.  It should 
   // be run each time before the FB_EventSummation blocks.
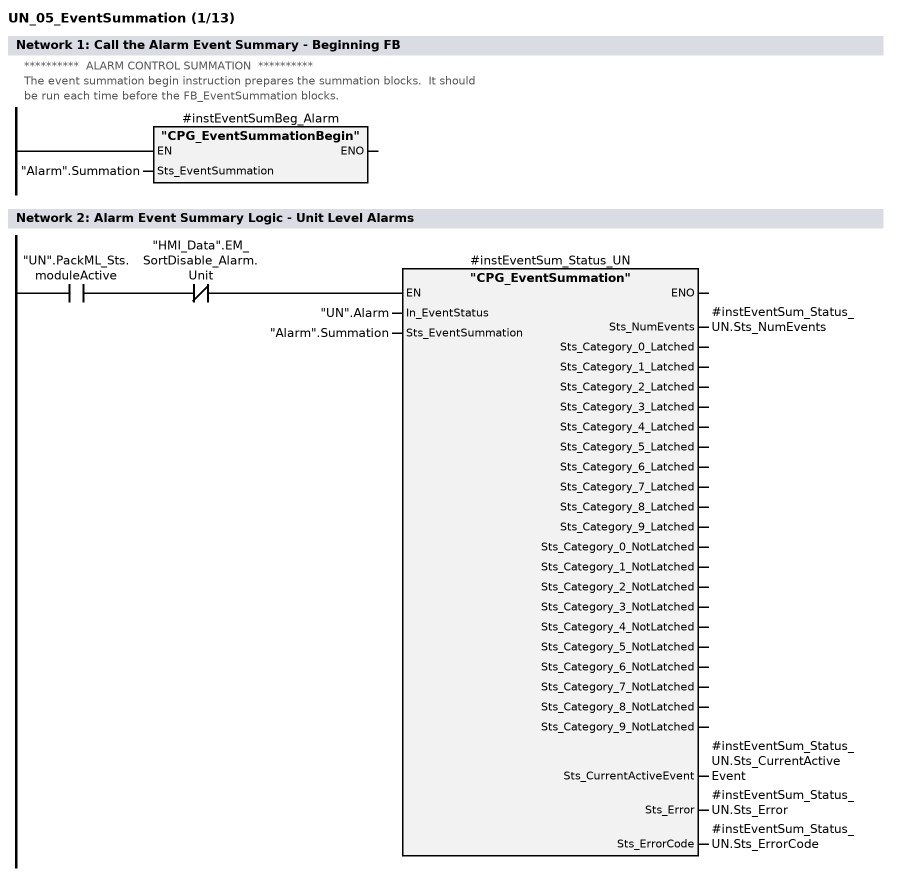
   RUNG wire#powerrail
      #instEventSumBeg_Alarm(Sts_EventSummation := "Alarm".Summation)
   END_RUNG
   // the same network as SCL:
   #instEventSumBeg_Alarm(Sts_EventSummation := "Alarm".Summation);   // "CPG_EventSummationBegin"
END_REGION

REGION Network 2: Alarm Event Summary Logic - Unit Level Alarms
   RUNG wire#powerrail
      Contact( "UN".PackML_Sts.moduleActive )
      I_Contact( "HMI_Data".EM_SortDisable_Alarm.Unit )
      #instEventSum_Status_UN(In_EventStatus := "UN".Alarm, Sts_EventSummation := "Alarm".Summation, Sts_NumEvents => #instEventSum_Status_UN.Sts_NumEvents, Sts_Category_0_Latched =>, Sts_Category_1_Latched =>, Sts_Category_2_Latched =>, Sts_Category_3_Latched =>, Sts_Category_4_Latched =>, Sts_Category_5_Latched =>, Sts_Category_6_Latched =>, Sts_Category_7_Latched =>, Sts_Category_8_Latched =>, Sts_Category_9_Latched =>, Sts_Category_0_NotLatched =>, Sts_Category_1_NotLatched =>, Sts_Category_2_NotLatched =>, Sts_Category_3_NotLatched =>, Sts_Category_4_NotLatched =>, Sts_Category_5_NotLatched =>, Sts_Category_6_NotLatched =>, Sts_Category_7_NotLatched =>, Sts_Category_8_NotLatched =>, Sts_Category_9_NotLatched =>, Sts_CurrentActiveEvent => #instEventSum_Status_UN.Sts_CurrentActiveEvent, Sts_Error => #instEventSum_Status_UN.Sts_Error, Sts_ErrorCode => #instEventSum_Status_UN.Sts_ErrorCode)
   END_RUNG
   // the same network as SCL:
   IF "UN".PackML_Sts.moduleActive AND NOT "HMI_Data".EM_SortDisable_Alarm.Unit THEN
       #instEventSum_Status_UN(In_EventStatus := "UN".Alarm,   // "CPG_EventSummation"
                               Sts_EventSummation := "Alarm".Summation,
                               Sts_NumEvents => #instEventSum_Status_UN.Sts_NumEvents,
                               Sts_CurrentActiveEvent => #instEventSum_Status_UN.Sts_CurrentActiveEvent,
                               Sts_Error => #instEventSum_Status_UN.Sts_Error,
                               Sts_ErrorCode => #instEventSum_Status_UN.Sts_ErrorCode);
   END_IF;
END_REGION

REGION Network 3: Alarm Event Summary Logic - Equipment Module #00
   // This instance of the Event Sum (or Event Summation) is used to merge the events 
   // from EM0 into the larger Unit or UN evevts list.
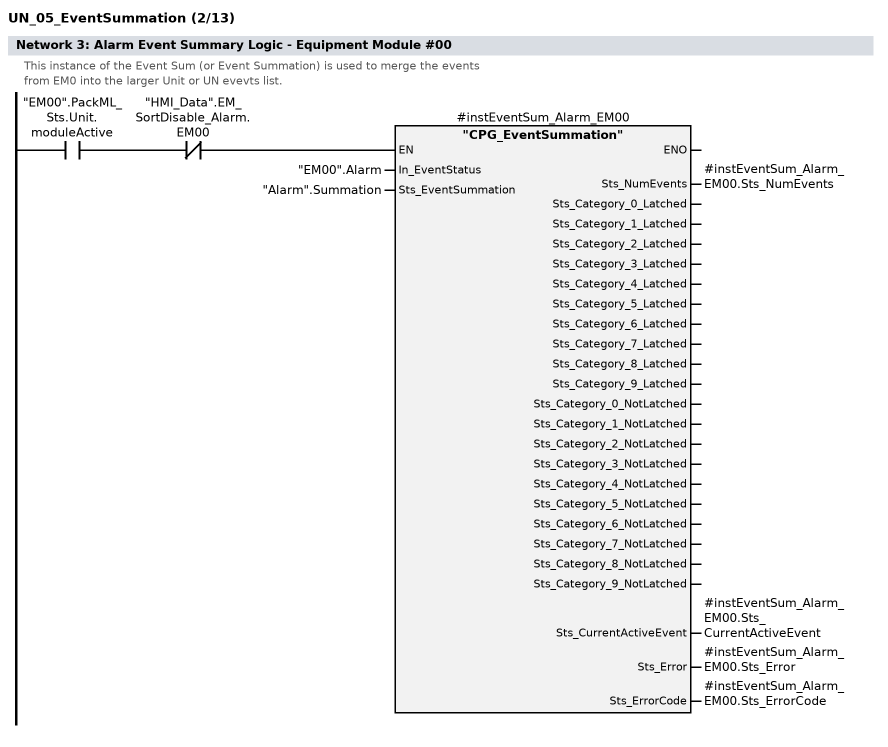
   RUNG wire#powerrail
      Contact( "EM00".PackML_Sts.Unit.moduleActive )
      I_Contact( "HMI_Data".EM_SortDisable_Alarm.EM00 )
      #instEventSum_Alarm_EM00(In_EventStatus := "EM00".Alarm, Sts_EventSummation := "Alarm".Summation, Sts_NumEvents => #instEventSum_Alarm_EM00.Sts_NumEvents, Sts_Category_0_Latched =>, Sts_Category_1_Latched =>, Sts_Category_2_Latched =>, Sts_Category_3_Latched =>, Sts_Category_4_Latched =>, Sts_Category_5_Latched =>, Sts_Category_6_Latched =>, Sts_Category_7_Latched =>, Sts_Category_8_Latched =>, Sts_Category_9_Latched =>, Sts_Category_0_NotLatched =>, Sts_Category_1_NotLatched =>, Sts_Category_2_NotLatched =>, Sts_Category_3_NotLatched =>, Sts_Category_4_NotLatched =>, Sts_Category_5_NotLatched =>, Sts_Category_6_NotLatched =>, Sts_Category_7_NotLatched =>, Sts_Category_8_NotLatched =>, Sts_Category_9_NotLatched =>, Sts_CurrentActiveEvent => #instEventSum_Alarm_EM00.Sts_CurrentActiveEvent, Sts_Error => #instEventSum_Alarm_EM00.Sts_Error, Sts_ErrorCode => #instEventSum_Alarm_EM00.Sts_ErrorCode)
   END_RUNG
   // the same network as SCL:
   IF "EM00".PackML_Sts.Unit.moduleActive AND NOT "HMI_Data".EM_SortDisable_Alarm.EM00 THEN
       #instEventSum_Alarm_EM00(In_EventStatus := "EM00".Alarm,   // "CPG_EventSummation"
                               Sts_EventSummation := "Alarm".Summation,
                               Sts_NumEvents => #instEventSum_Alarm_EM00.Sts_NumEvents,
                               Sts_CurrentActiveEvent => #instEventSum_Alarm_EM00.Sts_CurrentActiveEvent,
                               Sts_Error => #instEventSum_Alarm_EM00.Sts_Error,
                               Sts_ErrorCode => #instEventSum_Alarm_EM00.Sts_ErrorCode);
   END_IF;
END_REGION

REGION Network 4: Alarm Event Summary Logic - Equipment Module #01
   // This instance of the Event Sum (or Event Summation) is used to merge the events 
   // from EM01 into the larger Unit or UN evevts list.
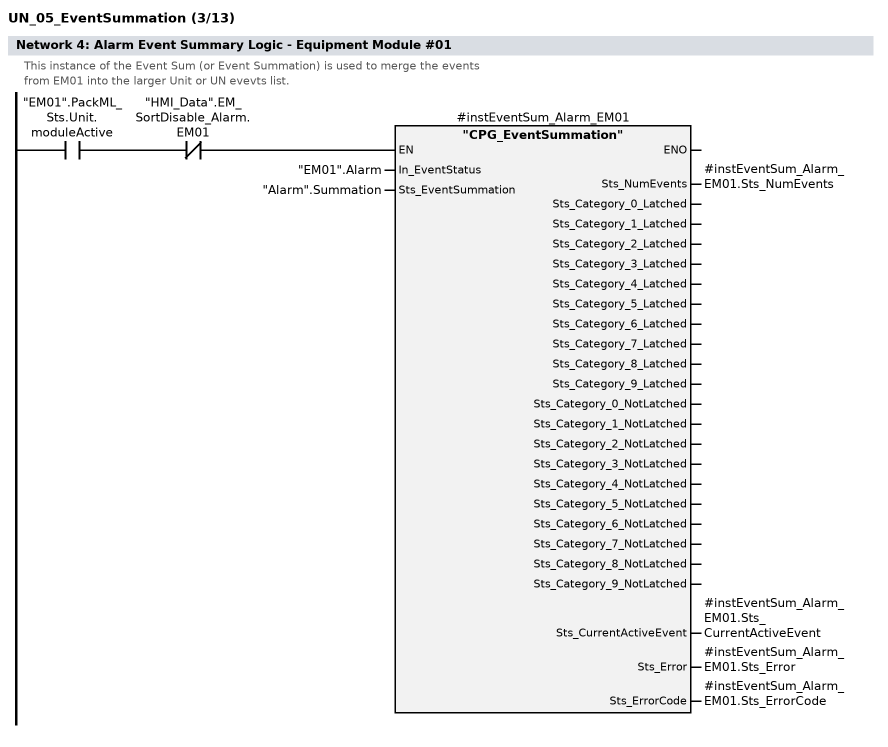
   RUNG wire#powerrail
      Contact( "EM01".PackML_Sts.Unit.moduleActive )
      I_Contact( "HMI_Data".EM_SortDisable_Alarm.EM01 )
      #instEventSum_Alarm_EM01(In_EventStatus := "EM01".Alarm, Sts_EventSummation := "Alarm".Summation, Sts_NumEvents => #instEventSum_Alarm_EM01.Sts_NumEvents, Sts_Category_0_Latched =>, Sts_Category_1_Latched =>, Sts_Category_2_Latched =>, Sts_Category_3_Latched =>, Sts_Category_4_Latched =>, Sts_Category_5_Latched =>, Sts_Category_6_Latched =>, Sts_Category_7_Latched =>, Sts_Category_8_Latched =>, Sts_Category_9_Latched =>, Sts_Category_0_NotLatched =>, Sts_Category_1_NotLatched =>, Sts_Category_2_NotLatched =>, Sts_Category_3_NotLatched =>, Sts_Category_4_NotLatched =>, Sts_Category_5_NotLatched =>, Sts_Category_6_NotLatched =>, Sts_Category_7_NotLatched =>, Sts_Category_8_NotLatched =>, Sts_Category_9_NotLatched =>, Sts_CurrentActiveEvent => #instEventSum_Alarm_EM01.Sts_CurrentActiveEvent, Sts_Error => #instEventSum_Alarm_EM01.Sts_Error, Sts_ErrorCode => #instEventSum_Alarm_EM01.Sts_ErrorCode)
   END_RUNG
   // the same network as SCL:
   IF "EM01".PackML_Sts.Unit.moduleActive AND NOT "HMI_Data".EM_SortDisable_Alarm.EM01 THEN
       #instEventSum_Alarm_EM01(In_EventStatus := "EM01".Alarm,   // "CPG_EventSummation"
                               Sts_EventSummation := "Alarm".Summation,
                               Sts_NumEvents => #instEventSum_Alarm_EM01.Sts_NumEvents,
                               Sts_CurrentActiveEvent => #instEventSum_Alarm_EM01.Sts_CurrentActiveEvent,
                               Sts_Error => #instEventSum_Alarm_EM01.Sts_Error,
                               Sts_ErrorCode => #instEventSum_Alarm_EM01.Sts_ErrorCode);
   END_IF;
END_REGION

REGION Network 5: Alarm Event Summary Logic - Equipment Module #02
   // This instance of the Event Sum (or Event Summation) is used to merge the events 
   // from EM01 into the larger Unit or UN evevts list.
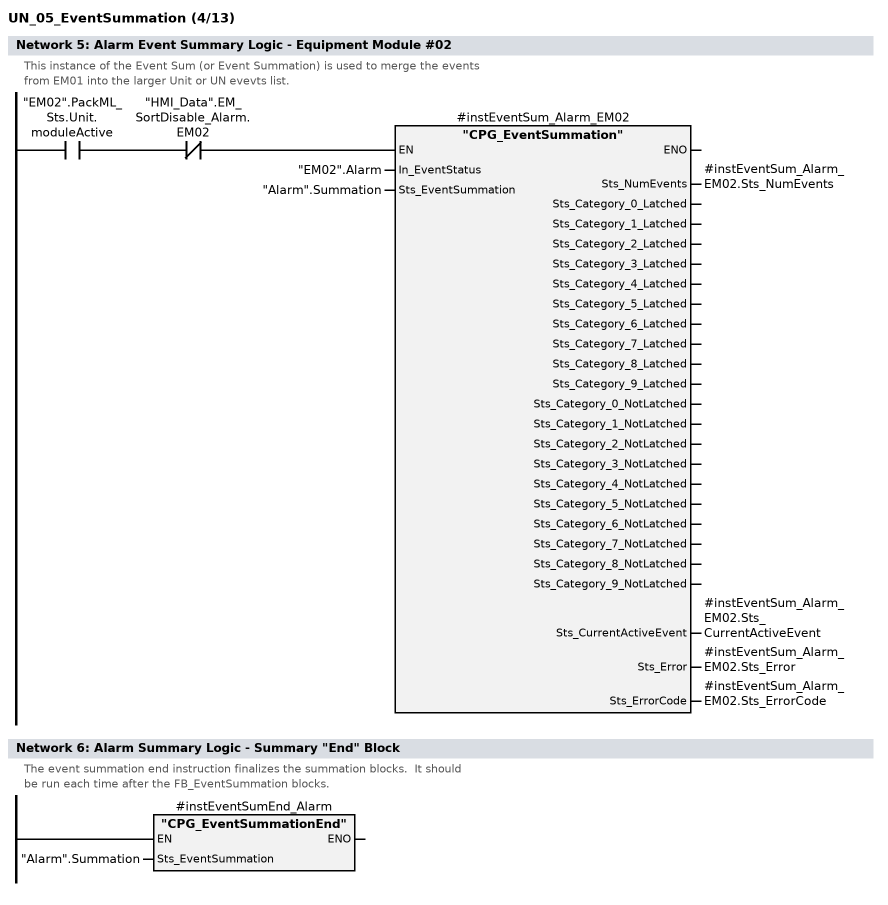
   RUNG wire#powerrail
      Contact( "EM02".PackML_Sts.Unit.moduleActive )
      I_Contact( "HMI_Data".EM_SortDisable_Alarm.EM02 )
      #instEventSum_Alarm_EM02(In_EventStatus := "EM02".Alarm, Sts_EventSummation := "Alarm".Summation, Sts_NumEvents => #instEventSum_Alarm_EM02.Sts_NumEvents, Sts_Category_0_Latched =>, Sts_Category_1_Latched =>, Sts_Category_2_Latched =>, Sts_Category_3_Latched =>, Sts_Category_4_Latched =>, Sts_Category_5_Latched =>, Sts_Category_6_Latched =>, Sts_Category_7_Latched =>, Sts_Category_8_Latched =>, Sts_Category_9_Latched =>, Sts_Category_0_NotLatched =>, Sts_Category_1_NotLatched =>, Sts_Category_2_NotLatched =>, Sts_Category_3_NotLatched =>, Sts_Category_4_NotLatched =>, Sts_Category_5_NotLatched =>, Sts_Category_6_NotLatched =>, Sts_Category_7_NotLatched =>, Sts_Category_8_NotLatched =>, Sts_Category_9_NotLatched =>, Sts_CurrentActiveEvent => #instEventSum_Alarm_EM02.Sts_CurrentActiveEvent, Sts_Error => #instEventSum_Alarm_EM02.Sts_Error, Sts_ErrorCode => #instEventSum_Alarm_EM02.Sts_ErrorCode)
   END_RUNG
   // the same network as SCL:
   IF "EM02".PackML_Sts.Unit.moduleActive AND NOT "HMI_Data".EM_SortDisable_Alarm.EM02 THEN
       #instEventSum_Alarm_EM02(In_EventStatus := "EM02".Alarm,   // "CPG_EventSummation"
                               Sts_EventSummation := "Alarm".Summation,
                               Sts_NumEvents => #instEventSum_Alarm_EM02.Sts_NumEvents,
                               Sts_CurrentActiveEvent => #instEventSum_Alarm_EM02.Sts_CurrentActiveEvent,
                               Sts_Error => #instEventSum_Alarm_EM02.Sts_Error,
                               Sts_ErrorCode => #instEventSum_Alarm_EM02.Sts_ErrorCode);
   END_IF;
END_REGION

REGION Network 6: Alarm Summary Logic - Summary "End" Block
   // The event summation end instruction finalizes the summation blocks.  It should 
   // be run each time after the FB_EventSummation blocks.
   RUNG wire#powerrail
      #instEventSumEnd_Alarm(Sts_EventSummation := "Alarm".Summation)
   END_RUNG
   // the same network as SCL:
   #instEventSumEnd_Alarm(Sts_EventSummation := "Alarm".Summation);   // "CPG_EventSummationEnd"
END_REGION

REGION Network 7: Update Admin.Alarm information.
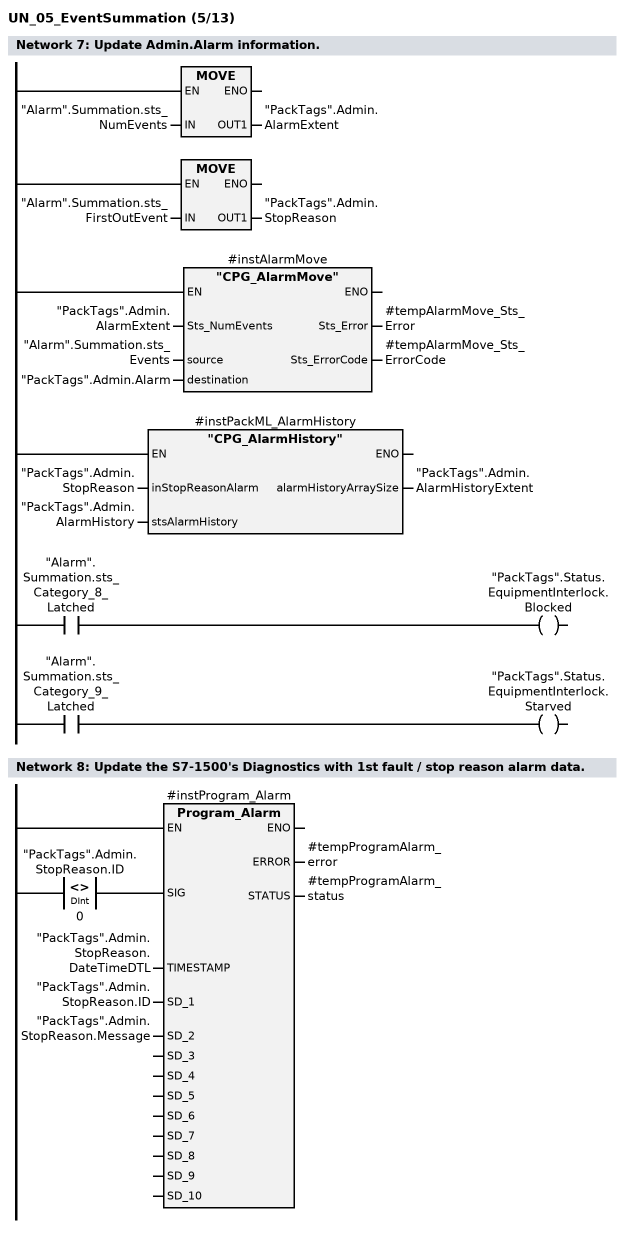
   RUNG wire#powerrail
      { S7_GenerateENO := "TRUE" } Move(in := "Alarm".Summation.sts_NumEvents, out1 => "PackTags".Admin.AlarmExtent)
   END_RUNG
   RUNG wire#powerrail
      Move(in := "Alarm".Summation.sts_FirstOutEvent, out1 => "PackTags".Admin.StopReason)
   END_RUNG
   RUNG wire#powerrail
      #instAlarmMove(Sts_NumEvents := "PackTags".Admin.AlarmExtent, source := "Alarm".Summation.sts_Events, destination := "PackTags".Admin.Alarm, Sts_Error => #tempAlarmMove_Sts_Error, Sts_ErrorCode => #tempAlarmMove_Sts_ErrorCode)
   END_RUNG
   RUNG wire#powerrail
      #instPackML_AlarmHistory(inStopReasonAlarm := "PackTags".Admin.StopReason, stsAlarmHistory := "PackTags".Admin.AlarmHistory, alarmHistoryArraySize => "PackTags".Admin.AlarmHistoryExtent)
   END_RUNG
   RUNG wire#powerrail
      Contact( "Alarm".Summation.sts_Category_8_Latched )
      Coil( "PackTags".Status.EquipmentInterlock.Blocked )
   END_RUNG
   RUNG wire#powerrail
      Contact( "Alarm".Summation.sts_Category_9_Latched )
      Coil( "PackTags".Status.EquipmentInterlock.Starved )
   END_RUNG
   // the same network as SCL:
   "PackTags".Admin.AlarmExtent := "Alarm".Summation.sts_NumEvents;
   "PackTags".Admin.StopReason := "Alarm".Summation.sts_FirstOutEvent;
   #instAlarmMove(Sts_NumEvents := "PackTags".Admin.AlarmExtent,   // "CPG_AlarmMove"
                  source := "Alarm".Summation.sts_Events,
                  destination := "PackTags".Admin.Alarm,
                  Sts_Error => #tempAlarmMove_Sts_Error,
                  Sts_ErrorCode => #tempAlarmMove_Sts_ErrorCode);
   #instPackML_AlarmHistory(inStopReasonAlarm := "PackTags".Admin.StopReason,   // "CPG_AlarmHistory"
                           stsAlarmHistory := "PackTags".Admin.AlarmHistory,
                           alarmHistoryArraySize => "PackTags".Admin.AlarmHistoryExtent);
   "PackTags".Status.EquipmentInterlock.Blocked := "Alarm".Summation.sts_Category_8_Latched;
   "PackTags".Status.EquipmentInterlock.Starved := "Alarm".Summation.sts_Category_9_Latched;
END_REGION

REGION Network 8: Update the S7-1500's Diagnostics with 1st fault / stop reason alarm data.
   RUNG wire#powerrail
      #instProgram_Alarm.Program_Alarm(SIG := wire#w1, TIMESTAMP := "PackTags".Admin.StopReason.DateTimeDTL, SD_1 := "PackTags".Admin.StopReason.ID, SD_2 := "PackTags".Admin.StopReason.Message, SD_3 :=, SD_4 :=, SD_5 :=, SD_6 :=, SD_7 :=, SD_8 :=, SD_9 :=, SD_10 :=, Error => #tempProgramAlarm_error, Status => #tempProgramAlarm_status)
   END_RUNG
   RUNG wire#powerrail
      { S7_Templates := "SrcType := DInt" } NE_Contact(in1 := "PackTags".Admin.StopReason.ID, in2 := 0)
   END_RUNG wire#w1
   // the same network as SCL:
   #instProgram_Alarm(SIG := "PackTags".Admin.StopReason.ID <> 0,   // Program_Alarm
                      TIMESTAMP := "PackTags".Admin.StopReason.DateTimeDTL,
                      SD_1 := "PackTags".Admin.StopReason.ID,
                      SD_2 := "PackTags".Admin.StopReason.Message,
                      Error => #tempProgramAlarm_error,
                      Status => #tempProgramAlarm_status);
END_REGION

REGION Network 9: Event Sort Filter logic - Alarms
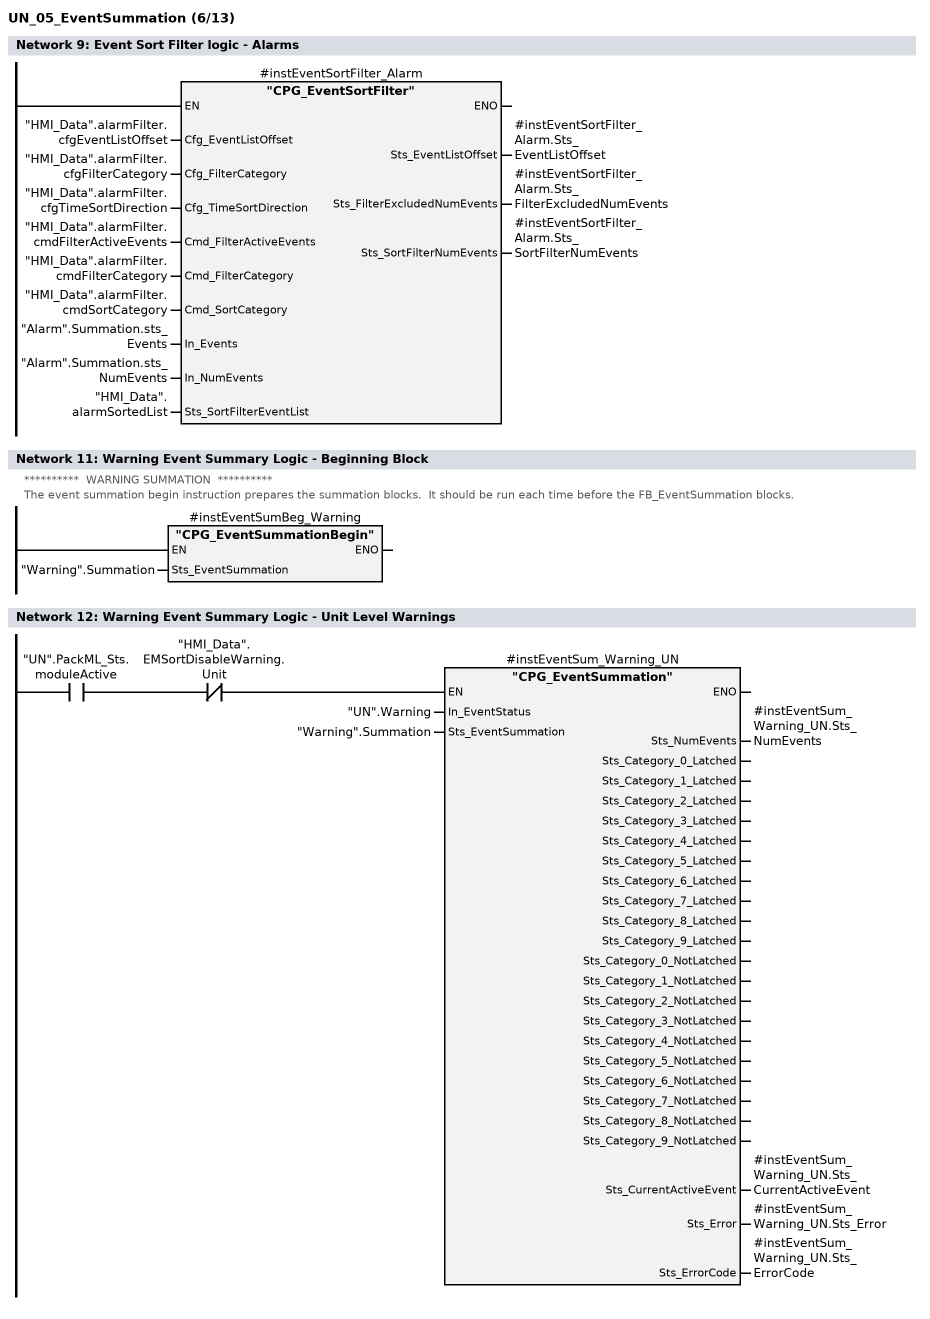
   RUNG wire#powerrail
      #instEventSortFilter_Alarm(Cfg_EventListOffset := "HMI_Data".alarmFilter.cfgEventListOffset, Cfg_FilterCategory := "HMI_Data".alarmFilter.cfgFilterCategory, Cfg_TimeSortDirection := "HMI_Data".alarmFilter.cfgTimeSortDirection, Cmd_FilterActiveEvents := "HMI_Data".alarmFilter.cmdFilterActiveEvents, Cmd_FilterCategory := "HMI_Data".alarmFilter.cmdFilterCategory, Cmd_SortCategory := "HMI_Data".alarmFilter.cmdSortCategory, In_Events := "Alarm".Summation.sts_Events, In_NumEvents := "Alarm".Summation.sts_NumEvents, Sts_SortFilterEventList := "HMI_Data".alarmSortedList, Sts_EventListOffset => #instEventSortFilter_Alarm.Sts_EventListOffset, Sts_FilterExcludedNumEvents => #instEventSortFilter_Alarm.Sts_FilterExcludedNumEvents, Sts_SortFilterNumEvents => #instEventSortFilter_Alarm.Sts_SortFilterNumEvents)
   END_RUNG
   // the same network as SCL:
   #instEventSortFilter_Alarm(Cfg_EventListOffset := "HMI_Data".alarmFilter.cfgEventListOffset,   // "CPG_EventSortFilter"
                           Cfg_FilterCategory := "HMI_Data".alarmFilter.cfgFilterCategory,
                           Cfg_TimeSortDirection := "HMI_Data".alarmFilter.cfgTimeSortDirection,
                           Cmd_FilterActiveEvents := "HMI_Data".alarmFilter.cmdFilterActiveEvents,
                           Cmd_FilterCategory := "HMI_Data".alarmFilter.cmdFilterCategory,
                           Cmd_SortCategory := "HMI_Data".alarmFilter.cmdSortCategory,
                           In_Events := "Alarm".Summation.sts_Events,
                           In_NumEvents := "Alarm".Summation.sts_NumEvents,
                           Sts_SortFilterEventList := "HMI_Data".alarmSortedList,
                           Sts_EventListOffset => #instEventSortFilter_Alarm.Sts_EventListOffset,
                           Sts_FilterExcludedNumEvents => #instEventSortFilter_Alarm.Sts_FilterExcludedNumEvents,
                           Sts_SortFilterNumEvents => #instEventSortFilter_Alarm.Sts_SortFilterNumEvents);
END_REGION

REGION Network 10: *** Beging the WARNING area ****
END_REGION

REGION Network 11: Warning Event Summary Logic - Beginning Block
   // **********  WARNING SUMMATION  **********
   //  
   // The event summation begin instruction prepares the summation blocks.  It should be run each time before the FB_EventSummation blocks.
   RUNG wire#powerrail
      #instEventSumBeg_Warning(Sts_EventSummation := "Warning".Summation)
   END_RUNG
   // the same network as SCL:
   #instEventSumBeg_Warning(Sts_EventSummation := "Warning".Summation);   // "CPG_EventSummationBegin"
END_REGION

REGION Network 12: Warning Event Summary Logic - Unit Level Warnings
   RUNG wire#powerrail
      Contact( "UN".PackML_Sts.moduleActive )
      I_Contact( "HMI_Data".EMSortDisableWarning.Unit )
      #instEventSum_Warning_UN(In_EventStatus := "UN".Warning, Sts_EventSummation := "Warning".Summation, Sts_NumEvents => #instEventSum_Warning_UN.Sts_NumEvents, Sts_Category_0_Latched =>, Sts_Category_1_Latched =>, Sts_Category_2_Latched =>, Sts_Category_3_Latched =>, Sts_Category_4_Latched =>, Sts_Category_5_Latched =>, Sts_Category_6_Latched =>, Sts_Category_7_Latched =>, Sts_Category_8_Latched =>, Sts_Category_9_Latched =>, Sts_Category_0_NotLatched =>, Sts_Category_1_NotLatched =>, Sts_Category_2_NotLatched =>, Sts_Category_3_NotLatched =>, Sts_Category_4_NotLatched =>, Sts_Category_5_NotLatched =>, Sts_Category_6_NotLatched =>, Sts_Category_7_NotLatched =>, Sts_Category_8_NotLatched =>, Sts_Category_9_NotLatched =>, Sts_CurrentActiveEvent => #instEventSum_Warning_UN.Sts_CurrentActiveEvent, Sts_Error => #instEventSum_Warning_UN.Sts_Error, Sts_ErrorCode => #instEventSum_Warning_UN.Sts_ErrorCode)
   END_RUNG
   // the same network as SCL:
   IF "UN".PackML_Sts.moduleActive AND NOT "HMI_Data".EMSortDisableWarning.Unit THEN
       #instEventSum_Warning_UN(In_EventStatus := "UN".Warning,   // "CPG_EventSummation"
                               Sts_EventSummation := "Warning".Summation,
                               Sts_NumEvents => #instEventSum_Warning_UN.Sts_NumEvents,
                               Sts_CurrentActiveEvent => #instEventSum_Warning_UN.Sts_CurrentActiveEvent,
                               Sts_Error => #instEventSum_Warning_UN.Sts_Error,
                               Sts_ErrorCode => #instEventSum_Warning_UN.Sts_ErrorCode);
   END_IF;
END_REGION

REGION Network 13: Warning Event Summary Logic - Equipment Module #00
   // This instance of the Event Sum (or Event Summation) is used to merge the events 
   // from EM0 into the larger Unit or UN evevts list.
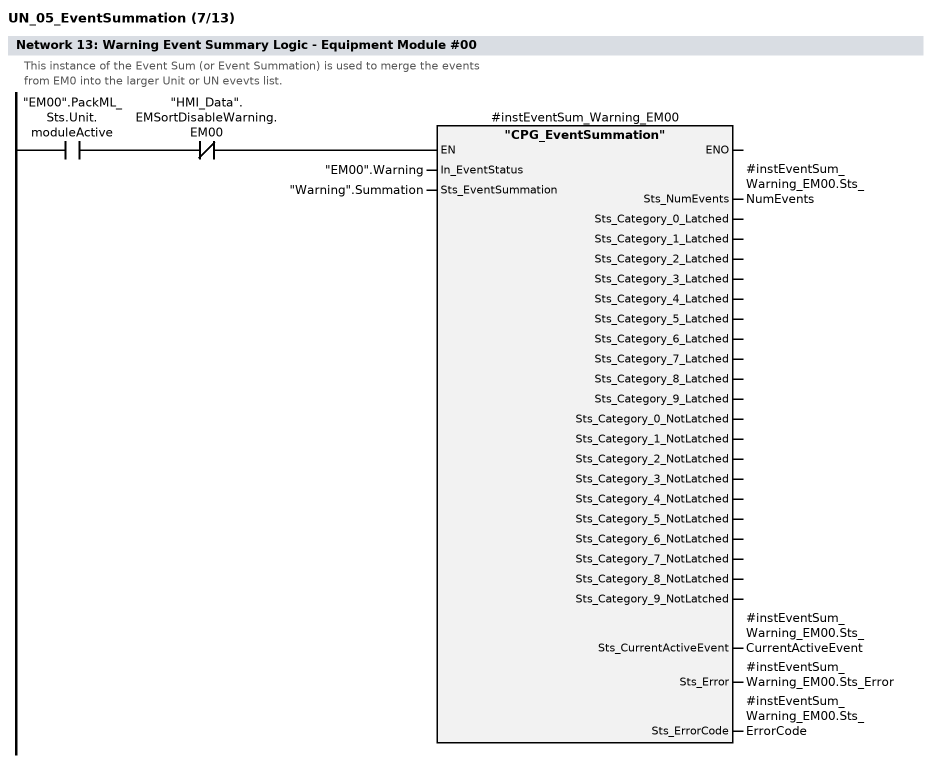
   RUNG wire#powerrail
      Contact( "EM00".PackML_Sts.Unit.moduleActive )
      I_Contact( "HMI_Data".EMSortDisableWarning.EM00 )
      #instEventSum_Warning_EM00(In_EventStatus := "EM00".Warning, Sts_EventSummation := "Warning".Summation, Sts_NumEvents => #instEventSum_Warning_EM00.Sts_NumEvents, Sts_Category_0_Latched =>, Sts_Category_1_Latched =>, Sts_Category_2_Latched =>, Sts_Category_3_Latched =>, Sts_Category_4_Latched =>, Sts_Category_5_Latched =>, Sts_Category_6_Latched =>, Sts_Category_7_Latched =>, Sts_Category_8_Latched =>, Sts_Category_9_Latched =>, Sts_Category_0_NotLatched =>, Sts_Category_1_NotLatched =>, Sts_Category_2_NotLatched =>, Sts_Category_3_NotLatched =>, Sts_Category_4_NotLatched =>, Sts_Category_5_NotLatched =>, Sts_Category_6_NotLatched =>, Sts_Category_7_NotLatched =>, Sts_Category_8_NotLatched =>, Sts_Category_9_NotLatched =>, Sts_CurrentActiveEvent => #instEventSum_Warning_EM00.Sts_CurrentActiveEvent, Sts_Error => #instEventSum_Warning_EM00.Sts_Error, Sts_ErrorCode => #instEventSum_Warning_EM00.Sts_ErrorCode)
   END_RUNG
   // the same network as SCL:
   IF "EM00".PackML_Sts.Unit.moduleActive AND NOT "HMI_Data".EMSortDisableWarning.EM00 THEN
       #instEventSum_Warning_EM00(In_EventStatus := "EM00".Warning,   // "CPG_EventSummation"
                               Sts_EventSummation := "Warning".Summation,
                               Sts_NumEvents => #instEventSum_Warning_EM00.Sts_NumEvents,
                               Sts_CurrentActiveEvent => #instEventSum_Warning_EM00.Sts_CurrentActiveEvent,
                               Sts_Error => #instEventSum_Warning_EM00.Sts_Error,
                               Sts_ErrorCode => #instEventSum_Warning_EM00.Sts_ErrorCode);
   END_IF;
END_REGION

REGION Network 14: Warning Event Summary Logic - Equipment Module #01
   // This instance of the Event Sum (or Event Summation) is used to merge the events 
   // from EM1 into the larger Unit or UN evevts list.
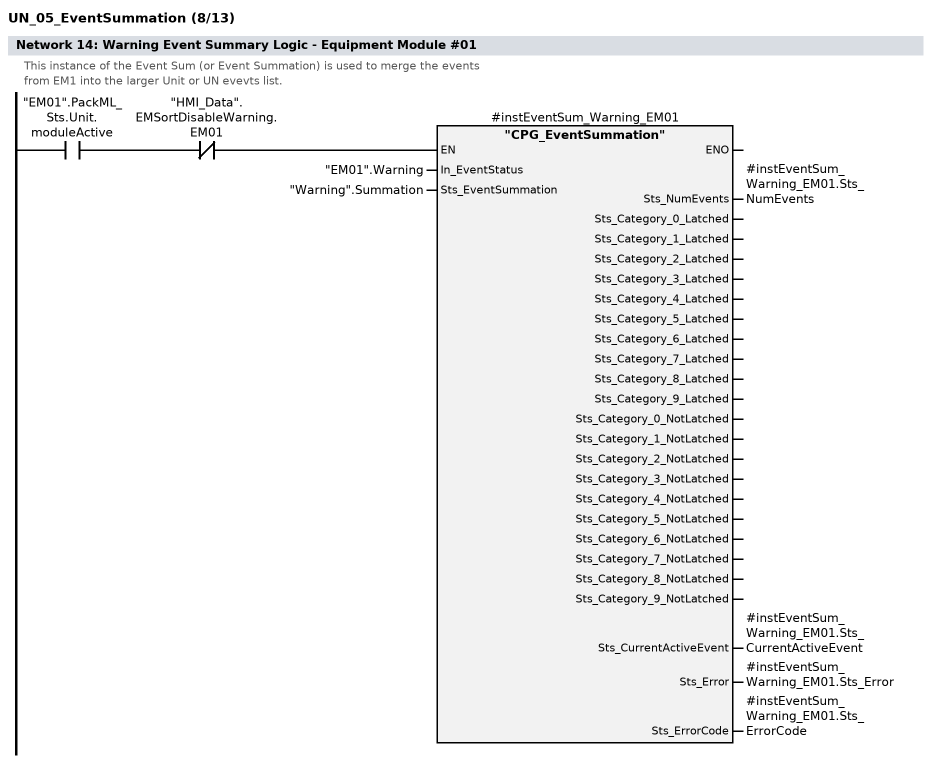
   RUNG wire#powerrail
      Contact( "EM01".PackML_Sts.Unit.moduleActive )
      I_Contact( "HMI_Data".EMSortDisableWarning.EM01 )
      #instEventSum_Warning_EM01(In_EventStatus := "EM01".Warning, Sts_EventSummation := "Warning".Summation, Sts_NumEvents => #instEventSum_Warning_EM01.Sts_NumEvents, Sts_Category_0_Latched =>, Sts_Category_1_Latched =>, Sts_Category_2_Latched =>, Sts_Category_3_Latched =>, Sts_Category_4_Latched =>, Sts_Category_5_Latched =>, Sts_Category_6_Latched =>, Sts_Category_7_Latched =>, Sts_Category_8_Latched =>, Sts_Category_9_Latched =>, Sts_Category_0_NotLatched =>, Sts_Category_1_NotLatched =>, Sts_Category_2_NotLatched =>, Sts_Category_3_NotLatched =>, Sts_Category_4_NotLatched =>, Sts_Category_5_NotLatched =>, Sts_Category_6_NotLatched =>, Sts_Category_7_NotLatched =>, Sts_Category_8_NotLatched =>, Sts_Category_9_NotLatched =>, Sts_CurrentActiveEvent => #instEventSum_Warning_EM01.Sts_CurrentActiveEvent, Sts_Error => #instEventSum_Warning_EM01.Sts_Error, Sts_ErrorCode => #instEventSum_Warning_EM01.Sts_ErrorCode)
   END_RUNG
   // the same network as SCL:
   IF "EM01".PackML_Sts.Unit.moduleActive AND NOT "HMI_Data".EMSortDisableWarning.EM01 THEN
       #instEventSum_Warning_EM01(In_EventStatus := "EM01".Warning,   // "CPG_EventSummation"
                               Sts_EventSummation := "Warning".Summation,
                               Sts_NumEvents => #instEventSum_Warning_EM01.Sts_NumEvents,
                               Sts_CurrentActiveEvent => #instEventSum_Warning_EM01.Sts_CurrentActiveEvent,
                               Sts_Error => #instEventSum_Warning_EM01.Sts_Error,
                               Sts_ErrorCode => #instEventSum_Warning_EM01.Sts_ErrorCode);
   END_IF;
END_REGION

REGION Network 15: Warning Event Summary Logic - Equipment Module #02
   // This instance of the Event Sum (or Event Summation) is used to merge the events 
   // from EM01 into the larger Unit or UN evevts list.
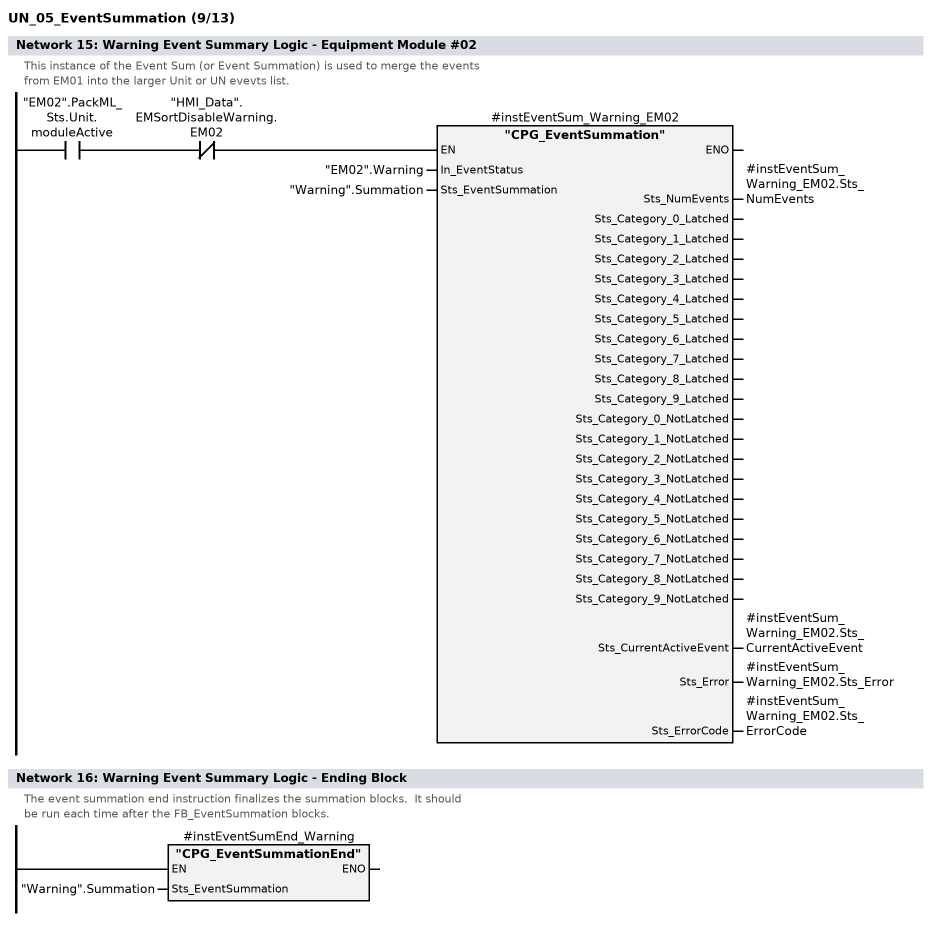
   RUNG wire#powerrail
      Contact( "EM02".PackML_Sts.Unit.moduleActive )
      I_Contact( "HMI_Data".EMSortDisableWarning.EM02 )
      #instEventSum_Warning_EM02(In_EventStatus := "EM02".Warning, Sts_EventSummation := "Warning".Summation, Sts_NumEvents => #instEventSum_Warning_EM02.Sts_NumEvents, Sts_Category_0_Latched =>, Sts_Category_1_Latched =>, Sts_Category_2_Latched =>, Sts_Category_3_Latched =>, Sts_Category_4_Latched =>, Sts_Category_5_Latched =>, Sts_Category_6_Latched =>, Sts_Category_7_Latched =>, Sts_Category_8_Latched =>, Sts_Category_9_Latched =>, Sts_Category_0_NotLatched =>, Sts_Category_1_NotLatched =>, Sts_Category_2_NotLatched =>, Sts_Category_3_NotLatched =>, Sts_Category_4_NotLatched =>, Sts_Category_5_NotLatched =>, Sts_Category_6_NotLatched =>, Sts_Category_7_NotLatched =>, Sts_Category_8_NotLatched =>, Sts_Category_9_NotLatched =>, Sts_CurrentActiveEvent => #instEventSum_Warning_EM02.Sts_CurrentActiveEvent, Sts_Error => #instEventSum_Warning_EM02.Sts_Error, Sts_ErrorCode => #instEventSum_Warning_EM02.Sts_ErrorCode)
   END_RUNG
   // the same network as SCL:
   IF "EM02".PackML_Sts.Unit.moduleActive AND NOT "HMI_Data".EMSortDisableWarning.EM02 THEN
       #instEventSum_Warning_EM02(In_EventStatus := "EM02".Warning,   // "CPG_EventSummation"
                               Sts_EventSummation := "Warning".Summation,
                               Sts_NumEvents => #instEventSum_Warning_EM02.Sts_NumEvents,
                               Sts_CurrentActiveEvent => #instEventSum_Warning_EM02.Sts_CurrentActiveEvent,
                               Sts_Error => #instEventSum_Warning_EM02.Sts_Error,
                               Sts_ErrorCode => #instEventSum_Warning_EM02.Sts_ErrorCode);
   END_IF;
END_REGION

REGION Network 16: Warning Event Summary Logic - Ending Block
   // The event summation end instruction finalizes the summation blocks.  It should 
   // be run each time after the FB_EventSummation blocks.
   RUNG wire#powerrail
      #instEventSumEnd_Warning(Sts_EventSummation := "Warning".Summation)
   END_RUNG
   // the same network as SCL:
   #instEventSumEnd_Warning(Sts_EventSummation := "Warning".Summation);   // "CPG_EventSummationEnd"
END_REGION

REGION Network 17: Event Sort Filter logic - Warnings
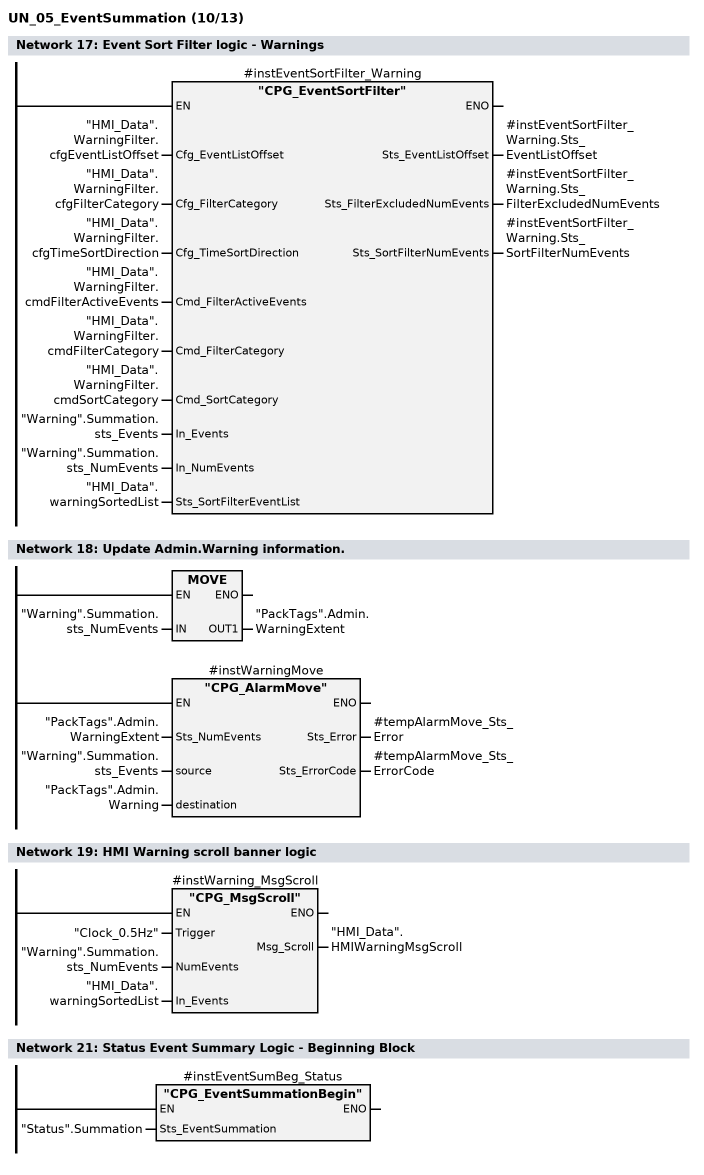
   RUNG wire#powerrail
      #instEventSortFilter_Warning(Cfg_EventListOffset := "HMI_Data".WarningFilter.cfgEventListOffset, Cfg_FilterCategory := "HMI_Data".WarningFilter.cfgFilterCategory, Cfg_TimeSortDirection := "HMI_Data".WarningFilter.cfgTimeSortDirection, Cmd_FilterActiveEvents := "HMI_Data".WarningFilter.cmdFilterActiveEvents, Cmd_FilterCategory := "HMI_Data".WarningFilter.cmdFilterCategory, Cmd_SortCategory := "HMI_Data".WarningFilter.cmdSortCategory, In_Events := "Warning".Summation.sts_Events, In_NumEvents := "Warning".Summation.sts_NumEvents, Sts_SortFilterEventList := "HMI_Data".warningSortedList, Sts_EventListOffset => #instEventSortFilter_Warning.Sts_EventListOffset, Sts_FilterExcludedNumEvents => #instEventSortFilter_Warning.Sts_FilterExcludedNumEvents, Sts_SortFilterNumEvents => #instEventSortFilter_Warning.Sts_SortFilterNumEvents)
   END_RUNG
   // the same network as SCL:
   #instEventSortFilter_Warning(Cfg_EventListOffset := "HMI_Data".WarningFilter.cfgEventListOffset,   // "CPG_EventSortFilter"
                           Cfg_FilterCategory := "HMI_Data".WarningFilter.cfgFilterCategory,
                           Cfg_TimeSortDirection := "HMI_Data".WarningFilter.cfgTimeSortDirection,
                           Cmd_FilterActiveEvents := "HMI_Data".WarningFilter.cmdFilterActiveEvents,
                           Cmd_FilterCategory := "HMI_Data".WarningFilter.cmdFilterCategory,
                           Cmd_SortCategory := "HMI_Data".WarningFilter.cmdSortCategory,
                           In_Events := "Warning".Summation.sts_Events,
                           In_NumEvents := "Warning".Summation.sts_NumEvents,
                           Sts_SortFilterEventList := "HMI_Data".warningSortedList,
                           Sts_EventListOffset => #instEventSortFilter_Warning.Sts_EventListOffset,
                           Sts_FilterExcludedNumEvents => #instEventSortFilter_Warning.Sts_FilterExcludedNumEvents,
                           Sts_SortFilterNumEvents => #instEventSortFilter_Warning.Sts_SortFilterNumEvents);
END_REGION

REGION Network 18: Update Admin.Warning information.
   RUNG wire#powerrail
      { S7_GenerateENO := "TRUE" } Move(in := "Warning".Summation.sts_NumEvents, out1 => "PackTags".Admin.WarningExtent)
   END_RUNG
   RUNG wire#powerrail
      #instWarningMove(Sts_NumEvents := "PackTags".Admin.WarningExtent, source := "Warning".Summation.sts_Events, destination := "PackTags".Admin.Warning, Sts_Error => #tempAlarmMove_Sts_Error, Sts_ErrorCode => #tempAlarmMove_Sts_ErrorCode)
   END_RUNG
   // the same network as SCL:
   "PackTags".Admin.WarningExtent := "Warning".Summation.sts_NumEvents;
   #instWarningMove(Sts_NumEvents := "PackTags".Admin.WarningExtent,   // "CPG_AlarmMove"
                    source := "Warning".Summation.sts_Events,
                    destination := "PackTags".Admin.Warning,
                    Sts_Error => #tempAlarmMove_Sts_Error,
                    Sts_ErrorCode => #tempAlarmMove_Sts_ErrorCode);
END_REGION

REGION Network 19: HMI Warning scroll banner logic
   RUNG wire#powerrail
      #instWarning_MsgScroll(Trigger := "Clock_0.5Hz", NumEvents := "Warning".Summation.sts_NumEvents, In_Events := "HMI_Data".warningSortedList, Msg_Scroll => "HMI_Data".HMIWarningMsgScroll)
   END_RUNG
   // the same network as SCL:
   #instWarning_MsgScroll(Trigger := "Clock_0.5Hz",   // "CPG_MsgScroll"
                          NumEvents := "Warning".Summation.sts_NumEvents,
                          In_Events := "HMI_Data".warningSortedList,
                          Msg_Scroll => "HMI_Data".HMIWarningMsgScroll);
END_REGION

REGION Network 20: *** Status Event Summation ***
END_REGION

REGION Network 21: Status Event Summary Logic - Beginning Block
   RUNG wire#powerrail
      #instEventSumBeg_Status(Sts_EventSummation := "Status".Summation)
   END_RUNG
   // the same network as SCL:
   #instEventSumBeg_Status(Sts_EventSummation := "Status".Summation);   // "CPG_EventSummationBegin"
END_REGION

REGION Network 22: Status Event Summary Logic - Unit
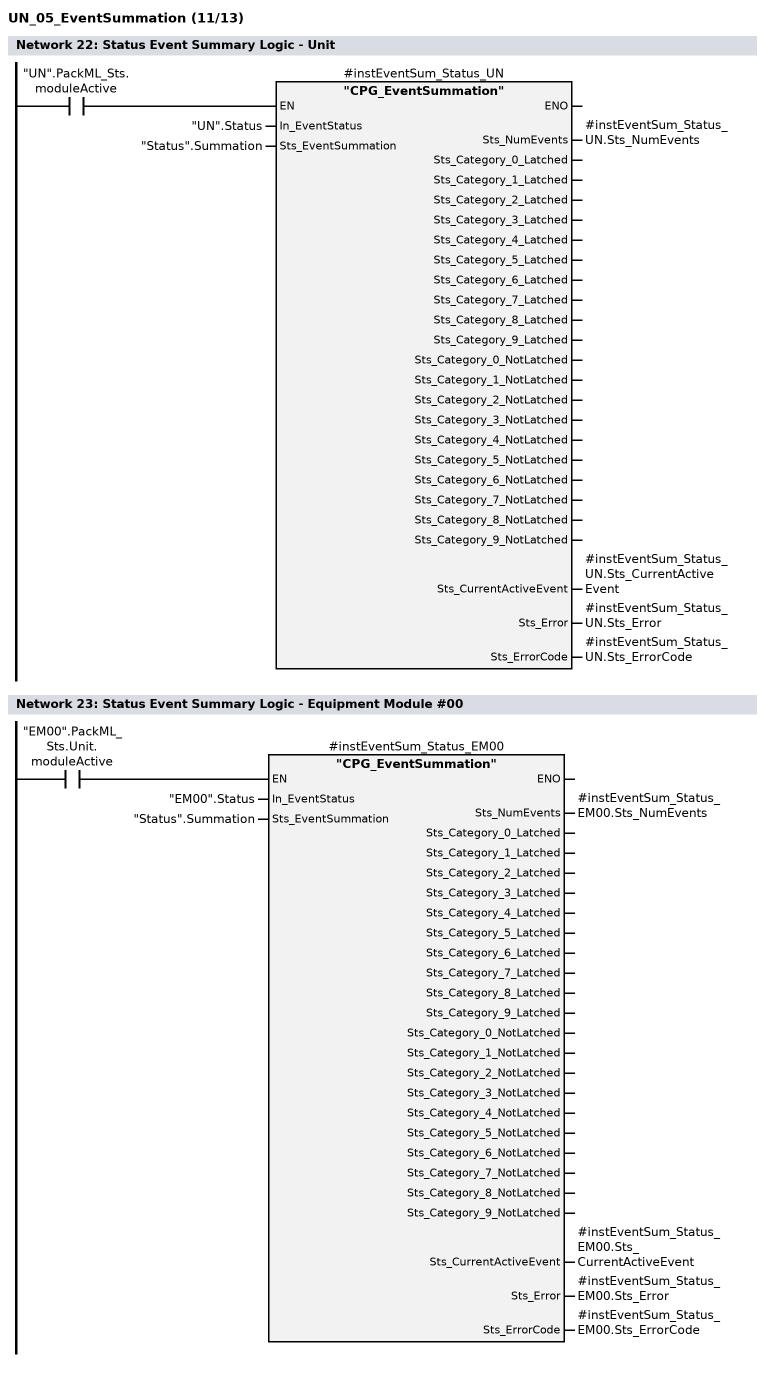
   RUNG wire#powerrail
      Contact( "UN".PackML_Sts.moduleActive )
      #instEventSum_Status_UN(In_EventStatus := "UN".Status, Sts_EventSummation := "Status".Summation, Sts_NumEvents => #instEventSum_Status_UN.Sts_NumEvents, Sts_Category_0_Latched =>, Sts_Category_1_Latched =>, Sts_Category_2_Latched =>, Sts_Category_3_Latched =>, Sts_Category_4_Latched =>, Sts_Category_5_Latched =>, Sts_Category_6_Latched =>, Sts_Category_7_Latched =>, Sts_Category_8_Latched =>, Sts_Category_9_Latched =>, Sts_Category_0_NotLatched =>, Sts_Category_1_NotLatched =>, Sts_Category_2_NotLatched =>, Sts_Category_3_NotLatched =>, Sts_Category_4_NotLatched =>, Sts_Category_5_NotLatched =>, Sts_Category_6_NotLatched =>, Sts_Category_7_NotLatched =>, Sts_Category_8_NotLatched =>, Sts_Category_9_NotLatched =>, Sts_CurrentActiveEvent => #instEventSum_Status_UN.Sts_CurrentActiveEvent, Sts_Error => #instEventSum_Status_UN.Sts_Error, Sts_ErrorCode => #instEventSum_Status_UN.Sts_ErrorCode)
   END_RUNG
   // the same network as SCL:
   IF "UN".PackML_Sts.moduleActive THEN
       #instEventSum_Status_UN(In_EventStatus := "UN".Status,   // "CPG_EventSummation"
                               Sts_EventSummation := "Status".Summation,
                               Sts_NumEvents => #instEventSum_Status_UN.Sts_NumEvents,
                               Sts_CurrentActiveEvent => #instEventSum_Status_UN.Sts_CurrentActiveEvent,
                               Sts_Error => #instEventSum_Status_UN.Sts_Error,
                               Sts_ErrorCode => #instEventSum_Status_UN.Sts_ErrorCode);
   END_IF;
END_REGION

REGION Network 23: Status Event Summary Logic - Equipment Module #00
   RUNG wire#powerrail
      Contact( "EM00".PackML_Sts.Unit.moduleActive )
      #instEventSum_Status_EM00(In_EventStatus := "EM00".Status, Sts_EventSummation := "Status".Summation, Sts_NumEvents => #instEventSum_Status_EM00.Sts_NumEvents, Sts_Category_0_Latched =>, Sts_Category_1_Latched =>, Sts_Category_2_Latched =>, Sts_Category_3_Latched =>, Sts_Category_4_Latched =>, Sts_Category_5_Latched =>, Sts_Category_6_Latched =>, Sts_Category_7_Latched =>, Sts_Category_8_Latched =>, Sts_Category_9_Latched =>, Sts_Category_0_NotLatched =>, Sts_Category_1_NotLatched =>, Sts_Category_2_NotLatched =>, Sts_Category_3_NotLatched =>, Sts_Category_4_NotLatched =>, Sts_Category_5_NotLatched =>, Sts_Category_6_NotLatched =>, Sts_Category_7_NotLatched =>, Sts_Category_8_NotLatched =>, Sts_Category_9_NotLatched =>, Sts_CurrentActiveEvent => #instEventSum_Status_EM00.Sts_CurrentActiveEvent, Sts_Error => #instEventSum_Status_EM00.Sts_Error, Sts_ErrorCode => #instEventSum_Status_EM00.Sts_ErrorCode)
   END_RUNG
   // the same network as SCL:
   IF "EM00".PackML_Sts.Unit.moduleActive THEN
       #instEventSum_Status_EM00(In_EventStatus := "EM00".Status,   // "CPG_EventSummation"
                               Sts_EventSummation := "Status".Summation,
                               Sts_NumEvents => #instEventSum_Status_EM00.Sts_NumEvents,
                               Sts_CurrentActiveEvent => #instEventSum_Status_EM00.Sts_CurrentActiveEvent,
                               Sts_Error => #instEventSum_Status_EM00.Sts_Error,
                               Sts_ErrorCode => #instEventSum_Status_EM00.Sts_ErrorCode);
   END_IF;
END_REGION

REGION Network 24: Status Event Summary Logic - Equipment Module #01
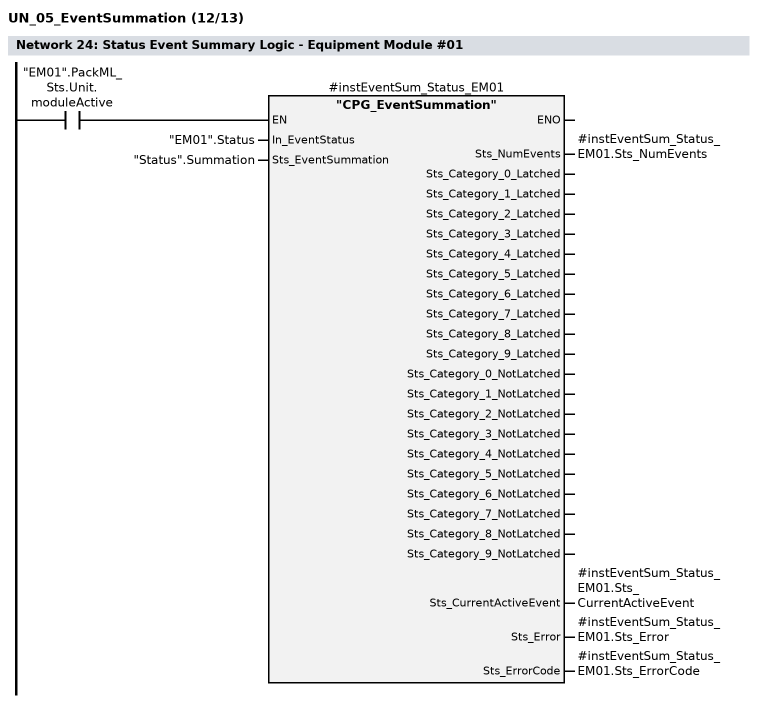
   RUNG wire#powerrail
      Contact( "EM01".PackML_Sts.Unit.moduleActive )
      #instEventSum_Status_EM01(In_EventStatus := "EM01".Status, Sts_EventSummation := "Status".Summation, Sts_NumEvents => #instEventSum_Status_EM01.Sts_NumEvents, Sts_Category_0_Latched =>, Sts_Category_1_Latched =>, Sts_Category_2_Latched =>, Sts_Category_3_Latched =>, Sts_Category_4_Latched =>, Sts_Category_5_Latched =>, Sts_Category_6_Latched =>, Sts_Category_7_Latched =>, Sts_Category_8_Latched =>, Sts_Category_9_Latched =>, Sts_Category_0_NotLatched =>, Sts_Category_1_NotLatched =>, Sts_Category_2_NotLatched =>, Sts_Category_3_NotLatched =>, Sts_Category_4_NotLatched =>, Sts_Category_5_NotLatched =>, Sts_Category_6_NotLatched =>, Sts_Category_7_NotLatched =>, Sts_Category_8_NotLatched =>, Sts_Category_9_NotLatched =>, Sts_CurrentActiveEvent => #instEventSum_Status_EM01.Sts_CurrentActiveEvent, Sts_Error => #instEventSum_Status_EM01.Sts_Error, Sts_ErrorCode => #instEventSum_Status_EM01.Sts_ErrorCode)
   END_RUNG
   // the same network as SCL:
   IF "EM01".PackML_Sts.Unit.moduleActive THEN
       #instEventSum_Status_EM01(In_EventStatus := "EM01".Status,   // "CPG_EventSummation"
                               Sts_EventSummation := "Status".Summation,
                               Sts_NumEvents => #instEventSum_Status_EM01.Sts_NumEvents,
                               Sts_CurrentActiveEvent => #instEventSum_Status_EM01.Sts_CurrentActiveEvent,
                               Sts_Error => #instEventSum_Status_EM01.Sts_Error,
                               Sts_ErrorCode => #instEventSum_Status_EM01.Sts_ErrorCode);
   END_IF;
END_REGION

REGION Network 25: Status Event Summary Logic - Equipment Module #02
   // This instance of the Event Sum (or Event Summation) is used to merge the events 
   // from EM01 into the larger Unit or UN evevts list.
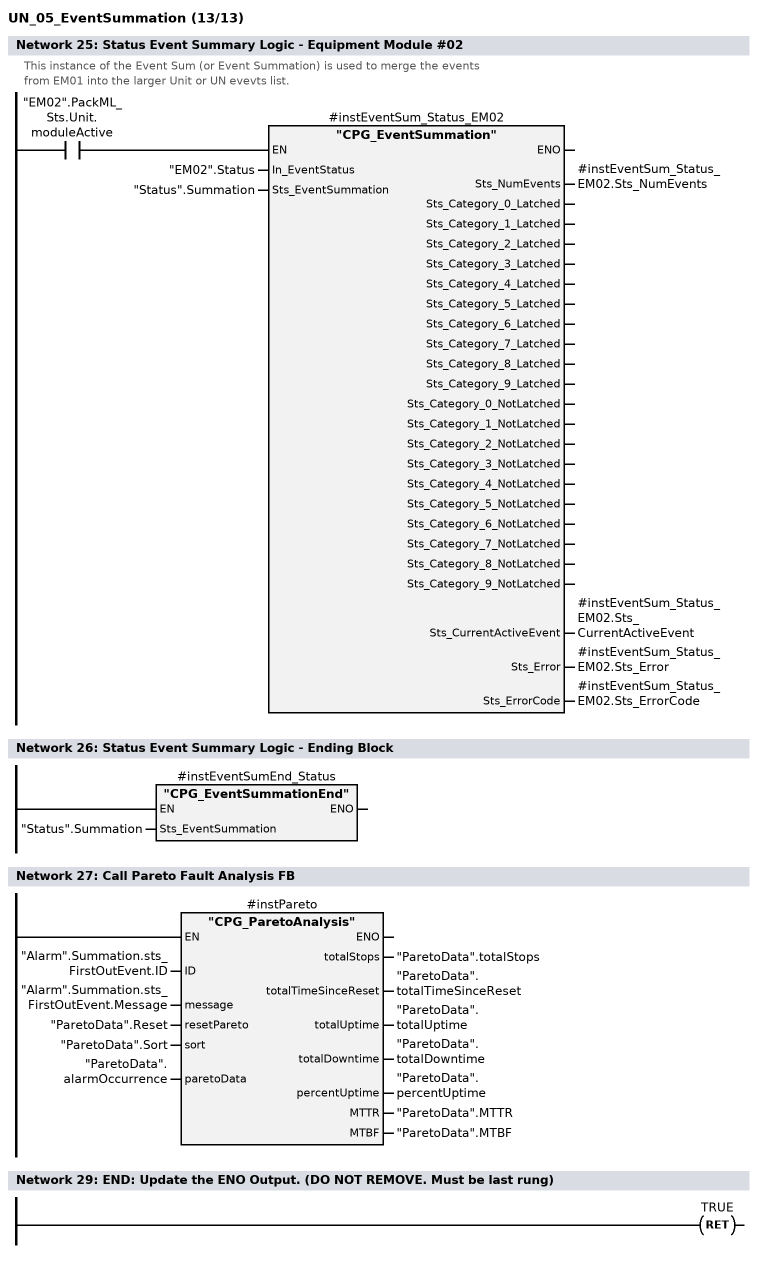
   RUNG wire#powerrail
      Contact( "EM02".PackML_Sts.Unit.moduleActive )
      #instEventSum_Status_EM02(In_EventStatus := "EM02".Status, Sts_EventSummation := "Status".Summation, Sts_NumEvents => #instEventSum_Status_EM02.Sts_NumEvents, Sts_Category_0_Latched =>, Sts_Category_1_Latched =>, Sts_Category_2_Latched =>, Sts_Category_3_Latched =>, Sts_Category_4_Latched =>, Sts_Category_5_Latched =>, Sts_Category_6_Latched =>, Sts_Category_7_Latched =>, Sts_Category_8_Latched =>, Sts_Category_9_Latched =>, Sts_Category_0_NotLatched =>, Sts_Category_1_NotLatched =>, Sts_Category_2_NotLatched =>, Sts_Category_3_NotLatched =>, Sts_Category_4_NotLatched =>, Sts_Category_5_NotLatched =>, Sts_Category_6_NotLatched =>, Sts_Category_7_NotLatched =>, Sts_Category_8_NotLatched =>, Sts_Category_9_NotLatched =>, Sts_CurrentActiveEvent => #instEventSum_Status_EM02.Sts_CurrentActiveEvent, Sts_Error => #instEventSum_Status_EM02.Sts_Error, Sts_ErrorCode => #instEventSum_Status_EM02.Sts_ErrorCode)
   END_RUNG
   // the same network as SCL:
   IF "EM02".PackML_Sts.Unit.moduleActive THEN
       #instEventSum_Status_EM02(In_EventStatus := "EM02".Status,   // "CPG_EventSummation"
                               Sts_EventSummation := "Status".Summation,
                               Sts_NumEvents => #instEventSum_Status_EM02.Sts_NumEvents,
                               Sts_CurrentActiveEvent => #instEventSum_Status_EM02.Sts_CurrentActiveEvent,
                               Sts_Error => #instEventSum_Status_EM02.Sts_Error,
                               Sts_ErrorCode => #instEventSum_Status_EM02.Sts_ErrorCode);
   END_IF;
END_REGION

REGION Network 26: Status Event Summary Logic - Ending Block
   RUNG wire#powerrail
      #instEventSumEnd_Status(Sts_EventSummation := "Status".Summation)
   END_RUNG
   // the same network as SCL:
   #instEventSumEnd_Status(Sts_EventSummation := "Status".Summation);   // "CPG_EventSummationEnd"
END_REGION

REGION Network 27: Call Pareto Fault Analysis FB
   RUNG wire#powerrail
      #instPareto(ID := "Alarm".Summation.sts_FirstOutEvent.ID, message := "Alarm".Summation.sts_FirstOutEvent.Message, resetPareto := "ParetoData".Reset, sort := "ParetoData".Sort, paretoData := "ParetoData".alarmOccurrence, totalStops => "ParetoData".totalStops, totalTimeSinceReset => "ParetoData".totalTimeSinceReset, totalUptime => "ParetoData".totalUptime, totalDowntime => "ParetoData".totalDowntime, percentUptime => "ParetoData".percentUptime, MTTR => "ParetoData".MTTR, MTBF => "ParetoData".MTBF)
   END_RUNG
   // the same network as SCL:
   #instPareto(ID := "Alarm".Summation.sts_FirstOutEvent.ID,   // "CPG_ParetoAnalysis"
               message := "Alarm".Summation.sts_FirstOutEvent.Message,
               resetPareto := "ParetoData".Reset,
               sort := "ParetoData".Sort,
               paretoData := "ParetoData".alarmOccurrence,
               totalStops => "ParetoData".totalStops,
               totalTimeSinceReset => "ParetoData".totalTimeSinceReset,
               totalUptime => "ParetoData".totalUptime,
               totalDowntime => "ParetoData".totalDowntime,
               percentUptime => "ParetoData".percentUptime,
               MTTR => "ParetoData".MTTR,
               MTBF => "ParetoData".MTBF);
END_REGION

REGION Network 28: HMI Warning scroll banner logic
END_REGION

REGION Network 29: END: Update the ENO Output. (DO NOT REMOVE. Must be last rung)
   RUNG wire#powerrail
      ReturnCoil( TRUE )
   END_RUNG
   // the same network as SCL:
   ENO := TRUE;
   RETURN;
END_REGION
END_FUNCTION_BLOCK

FUNCTION_BLOCK "CPG_EventSummationBegin"
TITLE = CPG_EventSummationBegin
{ S7_Optimized_Access := 'TRUE' }
AUTHOR : 'tech.team.motioncontrol@siemens.com'
FAMILY : CPG
VERSION : 1.0
//Support: tech.team.motioncontrol@siemens.com
   VAR_IN_OUT 
      Sts_EventSummation : "CPG_typeEventSummation";   // Working event list data section
   END_VAR

   VAR 
      statFirstScan { ExternalAccessible := 'False'; ExternalVisible := 'False'; ExternalWritable := 'False'} : Bool;   // 0=1st scan of FB; set to 1 after 1st FB scan...
      statIndex { ExternalAccessible := 'False'; ExternalVisible := 'False'; ExternalWritable := 'False'} : Int;   // temp value needed with FOR loop
      statZeroEvent { ExternalAccessible := 'False'; ExternalVisible := 'False'; ExternalWritable := 'False'} : "CPG_typeEvent";   // Null Event
   END_VAR


BEGIN
	//============================================================================================================
	// SIEMENS AG
	// (c)Copyright 2018 All Rights Reserved
	//------------------------------------------------------------------------------------------------------------
	// Project: CPG Template
	// Tested with: S7-1500 with FW version V2.1
	// Engineering: TIA Portal V14
	// Restrictions: ---
	// Requirements: S7-1500
	// Functionality:  Summarizes the "Data" from the equipment modules (from FB_EventManager) AND will create one list OF events FOR the unit machine.
	//                 It summarizes the data by finding the unit machine first out event and summarizes which category of events are active.
	//                 FB_EventSummationBegin initializes the summation, and FB_EventSummationEnd finalizes the summation.
	// Support: tech.team.motioncontrol@siemens.com
	//------------------------------------------------------------------------------------------------------------
	// Change log table:
	// Version       Date               Expert in charge    Changes applied
	//  01.00.00     01.01.2018         MP                  Initial Release & PackML V2.1  Renamed CPG V1.0
	//  01.01.00     29.05.2018         JP                  Adopted to styleguide
	//============================================================================================================
	// Function Block : CPG_EventSummationBegin
	//============================================================================================================
	
	
	
	// ===========================================================================
	// Begin the First Scan / Initialize logic section:
	IF #statFirstScan = FALSE THEN
	    // initialize & determine max array size
	    "CPG_ArrayLength"(arrayToBeSized := #Sts_EventSummation.sts_Events,
	                      arraySize => #Sts_EventSummation.wrk_EventArraySize);
	    
	    // initialize and clear the status events area
	           FOR #statIndex := 0 TO (#Sts_EventSummation.wrk_EventArraySize - 1) DO
	               #Sts_EventSummation.sts_Events[#statIndex] := #statZeroEvent;
	           END_FOR;
	    
	    #statFirstScan := TRUE;            // set the first scan bit 
	END_IF;
	// End of First Scan Section
	
	// Begin the LOGIC section:
	// Initialize the summation - This FB is to be called before the numerous "FB_PG_EventSum" calls.
	
	// Clear the first out event
	#Sts_EventSummation.sts_FirstOutEvent := #statZeroEvent;
	
	// Clear the first out event category arrays  
	FOR #statIndex := 0 TO 9 DO
	    #Sts_EventSummation.sts_FirstOutEventCat[#statIndex] := #statZeroEvent;
	END_FOR;
	
	// Determine the array size
	"CPG_ArrayLength"(arrayToBeSized := #Sts_EventSummation.sts_Events,
	                         arraySize => #Sts_EventSummation.wrk_EventArraySize);
	// Clear the number of events
	#Sts_EventSummation.sts_NumEvents := 0;            // set the number of events to 0.
	
	// Clear the output category status bits
	#Sts_EventSummation.wrk_Category_0_Latched := FALSE;
	#Sts_EventSummation.wrk_Category_1_Latched := FALSE;
	#Sts_EventSummation.wrk_Category_2_Latched := FALSE;
	#Sts_EventSummation.wrk_Category_3_Latched := FALSE;
	#Sts_EventSummation.wrk_Category_4_Latched := FALSE;
	#Sts_EventSummation.wrk_Category_5_Latched := FALSE;
	#Sts_EventSummation.wrk_Category_6_Latched := FALSE;
	#Sts_EventSummation.wrk_Category_7_Latched := FALSE;
	#Sts_EventSummation.wrk_Category_8_Latched := FALSE;
	#Sts_EventSummation.wrk_Category_9_Latched := FALSE;
	#Sts_EventSummation.wrk_Category_0_NotLatched := FALSE;
	#Sts_EventSummation.wrk_Category_1_NotLatched := FALSE;
	#Sts_EventSummation.wrk_Category_2_NotLatched := FALSE;
	#Sts_EventSummation.wrk_Category_3_NotLatched := FALSE;
	#Sts_EventSummation.wrk_Category_4_NotLatched := FALSE;
	#Sts_EventSummation.wrk_Category_5_NotLatched := FALSE;
	#Sts_EventSummation.wrk_Category_6_NotLatched := FALSE;
	#Sts_EventSummation.wrk_Category_7_NotLatched := FALSE;
	#Sts_EventSummation.wrk_Category_8_NotLatched := FALSE;
	#Sts_EventSummation.wrk_Category_9_NotLatched := FALSE;
	#Sts_EventSummation.wrk_CurrentActiveEvent := FALSE;
	
	//  -------------- END OF LOGIC -------------------------
	ENO := TRUE;   // Set the ENO output
	
END_FUNCTION_BLOCK

FUNCTION_BLOCK "CPG_EventSummation"
TITLE = CPG_EventSummation
{ S7_Optimized_Access := 'TRUE' }
AUTHOR : 'tech.team.motioncontrol@siemens.com'
FAMILY : CPG
VERSION : 1.0
//Support: tech.team.motioncontrol@siemens.com
   VAR_OUTPUT 
      Sts_NumEvents { ExternalAccessible := 'False'; ExternalVisible := 'False'; ExternalWritable := 'False'} : Int;   // Status - Number of active events
      Sts_Category_0_Latched { ExternalAccessible := 'False'; ExternalVisible := 'False'; ExternalWritable := 'False'; S7_HiddenAssignment := 'HideIfNoParamAssigned'} : Bool;   // Status - Latched Event - Cat. 0
      Sts_Category_1_Latched { ExternalAccessible := 'False'; ExternalVisible := 'False'; ExternalWritable := 'False'; S7_HiddenAssignment := 'HideIfNoParamAssigned'} : Bool;   // Status - Latched Event - Cat. 1
      Sts_Category_2_Latched { ExternalAccessible := 'False'; ExternalVisible := 'False'; ExternalWritable := 'False'; S7_HiddenAssignment := 'HideIfNoParamAssigned'} : Bool;   // Status - Latched Event - Cat. 2
      Sts_Category_3_Latched { ExternalAccessible := 'False'; ExternalVisible := 'False'; ExternalWritable := 'False'; S7_HiddenAssignment := 'HideIfNoParamAssigned'} : Bool;   // Status - Latched Event - Cat. 3
      Sts_Category_4_Latched { ExternalAccessible := 'False'; ExternalVisible := 'False'; ExternalWritable := 'False'; S7_HiddenAssignment := 'HideIfNoParamAssigned'} : Bool;   // Status - Latched Event - Cat. 4
      Sts_Category_5_Latched { ExternalAccessible := 'False'; ExternalVisible := 'False'; ExternalWritable := 'False'; S7_HiddenAssignment := 'HideIfNoParamAssigned'} : Bool;   // Status - Latched Event - Cat. 5
      Sts_Category_6_Latched { ExternalAccessible := 'False'; ExternalVisible := 'False'; ExternalWritable := 'False'; S7_HiddenAssignment := 'HideIfNoParamAssigned'} : Bool;   // Status - Latched Event - Cat. 6
      Sts_Category_7_Latched { ExternalAccessible := 'False'; ExternalVisible := 'False'; ExternalWritable := 'False'; S7_HiddenAssignment := 'HideIfNoParamAssigned'} : Bool;   // Status - Latched Event - Cat. 7
      Sts_Category_8_Latched { ExternalAccessible := 'False'; ExternalVisible := 'False'; ExternalWritable := 'False'; S7_HiddenAssignment := 'HideIfNoParamAssigned'} : Bool;   // Status - Latched Event - Cat. 8
      Sts_Category_9_Latched { ExternalAccessible := 'False'; ExternalVisible := 'False'; ExternalWritable := 'False'; S7_HiddenAssignment := 'HideIfNoParamAssigned'} : Bool;   // Status - Latched Event - Cat. 9
      Sts_Category_0_NotLatched { ExternalAccessible := 'False'; ExternalVisible := 'False'; ExternalWritable := 'False'; S7_HiddenAssignment := 'HideIfNoParamAssigned'} : Bool;   // Status - NotLatched (Active) Event - Cat. 0
      Sts_Category_1_NotLatched { ExternalAccessible := 'False'; ExternalVisible := 'False'; ExternalWritable := 'False'; S7_HiddenAssignment := 'HideIfNoParamAssigned'} : Bool;   // Status - NotLatched (Active) Event - Cat. 1
      Sts_Category_2_NotLatched { ExternalAccessible := 'False'; ExternalVisible := 'False'; ExternalWritable := 'False'; S7_HiddenAssignment := 'HideIfNoParamAssigned'} : Bool;   // Status - NotLatched (Active) Event - Cat. 2
      Sts_Category_3_NotLatched { ExternalAccessible := 'False'; ExternalVisible := 'False'; ExternalWritable := 'False'; S7_HiddenAssignment := 'HideIfNoParamAssigned'} : Bool;   // Status - NotLatched (Active) Event - Cat. 3
      Sts_Category_4_NotLatched { ExternalAccessible := 'False'; ExternalVisible := 'False'; ExternalWritable := 'False'; S7_HiddenAssignment := 'HideIfNoParamAssigned'} : Bool;   // Status - NotLatched (Active) Event - Cat. 4
      Sts_Category_5_NotLatched { ExternalAccessible := 'False'; ExternalVisible := 'False'; ExternalWritable := 'False'; S7_HiddenAssignment := 'HideIfNoParamAssigned'} : Bool;   // Status - NotLatched (Active) Event - Cat. 5
      Sts_Category_6_NotLatched { ExternalAccessible := 'False'; ExternalVisible := 'False'; ExternalWritable := 'False'; S7_HiddenAssignment := 'HideIfNoParamAssigned'} : Bool;   // Status - NotLatched (Active) Event - Cat. 6
      Sts_Category_7_NotLatched { ExternalAccessible := 'False'; ExternalVisible := 'False'; ExternalWritable := 'False'; S7_HiddenAssignment := 'HideIfNoParamAssigned'} : Bool;   // Status - NotLatched (Active) Event - Cat. 7
      Sts_Category_8_NotLatched { ExternalAccessible := 'False'; ExternalVisible := 'False'; ExternalWritable := 'False'; S7_HiddenAssignment := 'HideIfNoParamAssigned'} : Bool;   // Status - NotLatched (Active) Event - Cat. 8
      Sts_Category_9_NotLatched { ExternalAccessible := 'False'; ExternalVisible := 'False'; ExternalWritable := 'False'; S7_HiddenAssignment := 'HideIfNoParamAssigned'} : Bool;   // Status - NotLatched (Active) Event - Cat. 9
      Sts_CurrentActiveEvent { ExternalAccessible := 'False'; ExternalVisible := 'False'; ExternalWritable := 'False'} : Bool;   // Active Event Exists
      Sts_Error { ExternalAccessible := 'False'; ExternalVisible := 'False'; ExternalWritable := 'False'} : Bool;   // Error in FB
      Sts_ErrorCode { ExternalAccessible := 'False'; ExternalVisible := 'False'; ExternalWritable := 'False'} : DInt;   // Error Code
   END_VAR

   VAR_IN_OUT 
      In_EventStatus : "CPG_typeEventStatus";   // UDT of EventStatus
      Sts_EventSummation : "CPG_typeEventSummation";   // UDT of EventSummation
   END_VAR

   VAR 
      statFirstScan { ExternalAccessible := 'False'; ExternalVisible := 'False'; ExternalWritable := 'False'} : Bool;   // 0=1st scan of FB; set to 1 after 1st FB scan...
      statCfg_MaxEvents { ExternalAccessible := 'False'; ExternalVisible := 'False'; ExternalWritable := 'False'} : Int;   // number of events used from In_EventStatus array.
      statEventsRemaining { ExternalAccessible := 'False'; ExternalVisible := 'False'; ExternalWritable := 'False'} : Int;   // number of events remaining
      statCompareTrue { ExternalAccessible := 'False'; ExternalVisible := 'False'; ExternalWritable := 'False'} : Bool;   // Compare true?
      statIndex { ExternalAccessible := 'False'; ExternalVisible := 'False'; ExternalWritable := 'False'} : Int;   // Index counter
      statIndex1 { ExternalAccessible := 'False'; ExternalVisible := 'False'; ExternalWritable := 'False'} : Int;   // Index counter
      statIndex2 { ExternalAccessible := 'False'; ExternalVisible := 'False'; ExternalWritable := 'False'} : Int;   // Index counter
      statIndex3 { ExternalAccessible := 'False'; ExternalVisible := 'False'; ExternalWritable := 'False'} : Int;   // Index counter
      statIndex3a { ExternalAccessible := 'False'; ExternalVisible := 'False'; ExternalWritable := 'False'} : Int;   // Index counter
      statIndex3AOffset { ExternalAccessible := 'False'; ExternalVisible := 'False'; ExternalWritable := 'False'} : Int;   // Index counter
      statWriteData { ExternalAccessible := 'False'; ExternalVisible := 'False'; ExternalWritable := 'False'} : Bool;
   END_VAR

   VAR_TEMP 
      tempDTL1 {InstructionName := 'DTL'; LibVersion := '1.0'} : DTL;   // Temp Date & Time value as DTL format
      tempDTL2 {InstructionName := 'DTL'; LibVersion := '1.0'} : DTL;   // Temp Date & Time value as DTL format
      tempMoveBlkVariantRetVal : Int;   // temp return value for BlockMoveVariant
   END_VAR


BEGIN
	//============================================================================================================
	// SIEMENS AG
	// (c)Copyright 2018 All Rights Reserved
	//------------------------------------------------------------------------------------------------------------
	// Project: CPG Template
	// Tested with: S7-1500 with FW version V2.1
	// Engineering: TIA Portal V14
	// Restrictions: ---
	// Requirements: S7-1500
	// Functionality:  Summarizes the "Data" from the equipment modules (from FB_EventManager) AND will create one list OF events FOR the unit machine.
	//                 It summarizes the data by finding the unit machine first out event and summarizes which category of events are active.
	//                 CPG_EventSummationBegin initializes the summation, and CPG_EventSummationEnd finalizes the summation.
	// Support: tech.team.motioncontrol@siemens.com
	//------------------------------------------------------------------------------------------------------------
	// Change log table:
	// Version       Date               Expert in charge    Changes applied
	//  01.00.00     01.01.2018         MP                  Initial Release & PackML V2.1  Renamed CPG V1.0
	//  01.01.00     29.05.2018         JP                  Adopted to styleguide
	//============================================================================================================
	// Function Block : CPG_EventSummation
	//============================================================================================================
	
	
	// ===========================================================================
	//  BEGIN THE LOGIC SECTION:
	//  First scan section
	IF #statFirstScan = FALSE THEN
	    // initialize & determine max array size
	    // input array size (i.e. Array[0.."CPG_NO_STS_ELEMENTS_EVENT_STATUS"] of "typeCPG_Event")
	    "CPG_ArrayLength"(arrayToBeSized := #In_EventStatus.sts_Events,
	                      arraySize => #In_EventStatus.wrk_EventArraySize);
	    
	    "CPG_ArrayLength"(arrayToBeSized := #In_EventStatus.sts_Events,
	                      arraySize => #statCfg_MaxEvents);
	    
	    #statFirstScan := TRUE;            // set the first scan bit 
	END_IF;
	// End of First Scan Section
	
	
	// BEGIN THE MAIN LOGIC SECTION:
	#Sts_ErrorCode := 0;               // Set the status error code
	#statWriteData := FALSE;                // set write data to false
	
	// Set First Out Event
	#tempDTL1 := #In_EventStatus.sts_FirstOutEvent.DateTimeDTL;                  // Date & Time of Sts_FirstOutEventCat[index].TimeEvent
	
	IF #tempDTL1 <> DTL#1970-01-01-00:00:00.0 THEN                                  // is In_EventStatus.Sts_FirstOutEvent.TimeEvent <> 0?
	   #tempDTL2 := #Sts_EventSummation.sts_FirstOutEvent.DateTimeDTL;           // load the current value of the Sts_Eve..
	   #statWriteData := FALSE;                                                   // Reset the write data command.
	      IF #tempDTL2 = DTL#1970-01-01-00:00:00.0 THEN                             // is Sts_EventSummation.Sts_FirstOutEvent.TimeEvent = 0? 
	           #statWriteData := TRUE;
	      ELSIF #tempDTL1 < #tempDTL2 THEN                                   // is IN_event newer than Sts_event ?
	          #statWriteData := TRUE;
	      END_IF;     // End "IF (EQ_DT(DT1:=Sts_"
	END_IF;         // End "IF (NOT(EQ_DT(DT1:=In_Ev"
	
	IF #statWriteData THEN 
	   #Sts_EventSummation.sts_FirstOutEvent := #In_EventStatus.sts_FirstOutEvent;  // Update the First Fault event 
	END_IF; 
	
	// Set First Out Event by Category
	FOR #statIndex:= 0 TO 9 DO
	    
	    #tempDTL1:=#In_EventStatus.sts_FirstOutEventCat[#statIndex].DateTimeDTL;        // Date & Time of Sts_FirstOutEventCat[index].TimeEvent
	    
	    IF #tempDTL1 <> DTL#1970-01-01-00:00:00.0 THEN                                // is In_EventStatus.Sts_FirstOutEvent.TimeEvent <> 0?
	        
	        #tempDTL2:=#Sts_EventSummation.sts_FirstOutEventCat[#statIndex].DateTimeDTL;          // load the current value of the Sts_Eve..
	        #statWriteData:=0;                   // Reset the write data command.
	        
	        IF #tempDTL2 = DTL#1970-01-01-00:00:00.0 THEN                              // is Sts_EventSummation.Sts_FirstOutEvent.TimeEvent = 0? 
	            #statWriteData := TRUE;
	            
	        ELSIF #tempDTL1 < #tempDTL2 THEN   // is IN_event newer than Sts_event ?
	            
	            #statWriteData := TRUE;
	            
	        END_IF;     // End "IF (EQ_DT(DT1:=Sts_"
	    END_IF;         // End "IF (NOT(EQ_DT(DT1:=In_Ev"
	
	    IF #statWriteData THEN 
	        #Sts_EventSummation.sts_FirstOutEventCat[#statIndex] := #In_EventStatus.sts_FirstOutEventCat[#statIndex];  // Update the First Fault event 
	    END_IF; 
	END_FOR;     
	
	// ---------------------------------------------------------------
	// Set Active Events
	IF #In_EventStatus.sts_NumEvents > 0 THEN 
	    IF #In_EventStatus.sts_NumEvents > 0 AND #Sts_EventSummation.sts_NumEvents > 0 THEN
	        #statIndex1 := 0;
	        FOR #statIndex := 0 TO #In_EventStatus.sts_NumEvents - 1 DO
	            
	            WHILE #statIndex1 < #Sts_EventSummation.sts_NumEvents DO
	                
	                #statCompareTrue := FALSE;
	                #statIndex2 := 0;
	                
	                REPEAT
	                    IF #In_EventStatus.sts_Events[#statIndex].DateTimeDTL = #Sts_EventSummation.sts_Events[#statIndex1].DateTimeDTL THEN
	                        #statIndex2 := #statIndex2 + 1;
	                        
	                    ELSIF #In_EventStatus.sts_Events[#statIndex].DateTimeDTL < #Sts_EventSummation.sts_Events[#statIndex1].DateTimeDTL THEN
	                        #statCompareTrue := TRUE;
	                        
	                        EXIT;  // Exit the REPEAT loop
	                    ELSE
	                        EXIT;  // Exit the REPEAT loop
	                    END_IF;
	                UNTIL #statIndex2 = 7
	                END_REPEAT;
	                
	                IF #statCompareTrue THEN
	                    #statEventsRemaining := #Sts_EventSummation.sts_NumEvents - #statIndex1;
	                    #statIndex3AOffset := #statEventsRemaining - 1 + #statIndex1;
	                    
	                    FOR #statIndex3 := 0 TO #statEventsRemaining - 1 DO  // Backwards copy the data to shift it down to prevent the data from overwriting itself
	                        #statIndex3a := #statIndex3AOffset - #statIndex3;
	                        IF #statIndex3a + 1 < #Sts_EventSummation.wrk_EventArraySize THEN
	                            #Sts_EventSummation.sts_Events[#statIndex3a + 1] := #Sts_EventSummation.sts_Events[#statIndex3a];
	                        END_IF;
	                    END_FOR;
	                    
	                    #Sts_EventSummation.sts_Events[#statIndex1] := #In_EventStatus.sts_Events[#statIndex];
	                    
	                    IF #Sts_EventSummation.sts_NumEvents < #Sts_EventSummation.wrk_EventArraySize THEN
	                        #Sts_EventSummation.sts_NumEvents := #Sts_EventSummation.sts_NumEvents + 1;
	                        #statIndex1 := #statIndex1 + 1;
	                    END_IF;
	                    
	                    EXIT;  //Exit the WHILE loop
	                END_IF;
	                #statIndex1 := #statIndex1 + 1;
	            END_WHILE;
	            
	            // If the WHILE loop is done, then bulk copy the remaining events into the event summation array.
	            IF #statIndex1 = #Sts_EventSummation.sts_NumEvents THEN
	                #statEventsRemaining := #In_EventStatus.sts_NumEvents - #statIndex;
	                IF #statEventsRemaining + #Sts_EventSummation.sts_NumEvents > #Sts_EventSummation.wrk_EventArraySize THEN
	                    #statEventsRemaining := #Sts_EventSummation.wrk_EventArraySize - #Sts_EventSummation.sts_NumEvents;
	                    #Sts_ErrorCode := 1;
	                END_IF;
	                
	                IF #statEventsRemaining > 0 THEN
	                    #Sts_EventSummation.sts_Events[#statIndex1] := #In_EventStatus.sts_Events[#statIndex];
	                    #Sts_EventSummation.sts_NumEvents := #Sts_EventSummation.sts_NumEvents + #statEventsRemaining;
	                END_IF;
	                EXIT;  //Exit the FOR loop
	            END_IF;
	        END_FOR;
	    ELSIF #In_EventStatus.sts_NumEvents > 0 THEN
	        // The current event summation array is empty, so just bulk copy the data over.
	        IF #In_EventStatus.sts_NumEvents < #Sts_EventSummation.wrk_EventArraySize THEN
	            
